    {attribute	'TcLinkTo'	:=	'.Ctrl:=TIIB[LAMP_PNL2_EP15_EP6002-0002]^COM RxPDO-Map Outputs Channel 1^Ctrl;
                                 .D[0]:=TIIB[LAMP_PNL2_EP15_EP6002-0002]^COM RxPDO-Map Outputs Channel 1^Data Out 0;
                                 .D[1]:=TIIB[LAMP_PNL2_EP15_EP6002-0002]^COM RxPDO-Map Outputs Channel 1^Data Out 1;
                                 .D[2]:=TIIB[LAMP_PNL2_EP15_EP6002-0002]^COM RxPDO-Map Outputs Channel 1^Data Out 2;
                                 .D[3]:=TIIB[LAMP_PNL2_EP15_EP6002-0002]^COM RxPDO-Map Outputs Channel 1^Data Out 3;
                                 .D[4]:=TIIB[LAMP_PNL2_EP15_EP6002-0002]^COM RxPDO-Map Outputs Channel 1^Data Out 4;
                                 .D[5]:=TIIB[LAMP_PNL2_EP15_EP6002-0002]^COM RxPDO-Map Outputs Channel 1^Data Out 5;
                                 .D[6]:=TIIB[LAMP_PNL2_EP15_EP6002-0002]^COM RxPDO-Map Outputs Channel 1^Data Out 6;
                                 .D[7]:=TIIB[LAMP_PNL2_EP15_EP6002-0002]^COM RxPDO-Map Outputs Channel 1^Data Out 7;
                                 .D[8]:=TIIB[LAMP_PNL2_EP15_EP6002-0002]^COM RxPDO-Map Outputs Channel 1^Data Out 8;
                                 .D[9]:=TIIB[LAMP_PNL2_EP15_EP6002-0002]^COM RxPDO-Map Outputs Channel 1^Data Out 9;
                                 .D[10]:=TIIB[LAMP_PNL2_EP15_EP6002-0002]^COM RxPDO-Map Outputs Channel 1^Data Out 10;
                                 .D[11]:=TIIB[LAMP_PNL2_EP15_EP6002-0002]^COM RxPDO-Map Outputs Channel 1^Data Out 11;
                                 .D[12]:=TIIB[LAMP_PNL2_EP15_EP6002-0002]^COM RxPDO-Map Outputs Channel 1^Data Out 12;
                                 .D[13]:=TIIB[LAMP_PNL2_EP15_EP6002-0002]^COM RxPDO-Map Outputs Channel 1^Data Out 13;
                                 .D[14]:=TIIB[LAMP_PNL2_EP15_EP6002-0002]^COM RxPDO-Map Outputs Channel 1^Data Out 14;
                                 .D[15]:=TIIB[LAMP_PNL2_EP15_EP6002-0002]^COM RxPDO-Map Outputs Channel 1^Data Out 15;
                                 .D[16]:=TIIB[LAMP_PNL2_EP15_EP6002-0002]^COM RxPDO-Map Outputs Channel 1^Data Out 16;
                                 .D[17]:=TIIB[LAMP_PNL2_EP15_EP6002-0002]^COM RxPDO-Map Outputs Channel 1^Data Out 17;
                                 .D[18]:=TIIB[LAMP_PNL2_EP15_EP6002-0002]^COM RxPDO-Map Outputs Channel 1^Data Out 18;
                                 .D[19]:=TIIB[LAMP_PNL2_EP15_EP6002-0002]^COM RxPDO-Map Outputs Channel 1^Data Out 19;
                                 .D[20]:=TIIB[LAMP_PNL2_EP15_EP6002-0002]^COM RxPDO-Map Outputs Channel 1^Data Out 20;
                                 .D[21]:=TIIB[LAMP_PNL2_EP15_EP6002-0002]^COM RxPDO-Map Outputs Channel 1^Data Out 21;
    '}
    stComOut_LAMP_ROUGH_PTM_01		AT %Q*	:	EL6outData22B;
(*
    {attribute	'TcLinkTo'	:=	'.Status:=TIIB[LAMP_PNL2_EP15_EP6002-0002]^COM TxPDO-Map Inputs Channel 2^Status;
                                 .D[0]:=TIIB[LAMP_PNL2_EP15_EP6002-0002]^COM TxPDO-Map Inputs Channel 2^Data In 0;
                                 .D[1]:=TIIB[LAMP_PNL2_EP15_EP6002-0002]^COM TxPDO-Map Inputs Channel 2^Data In 1;
                                 .D[2]:=TIIB[LAMP_PNL2_EP15_EP6002-0002]^COM TxPDO-Map Inputs Channel 2^Data In 2;
                                 .D[3]:=TIIB[LAMP_PNL2_EP15_EP6002-0002]^COM TxPDO-Map Inputs Channel 2^Data In 3;
                                 .D[4]:=TIIB[LAMP_PNL2_EP15_EP6002-0002]^COM TxPDO-Map Inputs Channel 2^Data In 4;
                                 .D[5]:=TIIB[LAMP_PNL2_EP15_EP6002-0002]^COM TxPDO-Map Inputs Channel 2^Data In 5;
                                 .D[6]:=TIIB[LAMP_PNL2_EP15_EP6002-0002]^COM TxPDO-Map Inputs Channel 2^Data In 6;
                                 .D[7]:=TIIB[LAMP_PNL2_EP15_EP6002-0002]^COM TxPDO-Map Inputs Channel 2^Data In 7;
                                 .D[8]:=TIIB[LAMP_PNL2_EP15_EP6002-0002]^COM TxPDO-Map Inputs Channel 2^Data In 8;
                                 .D[9]:=TIIB[LAMP_PNL2_EP15_EP6002-0002]^COM TxPDO-Map Inputs Channel 2^Data In 9;
                                 .D[10]:=TIIB[LAMP_PNL2_EP15_EP6002-0002]^COM TxPDO-Map Inputs Channel 2^Data In 10;
                                 .D[11]:=TIIB[LAMP_PNL2_EP15_EP6002-0002]^COM TxPDO-Map Inputs Channel 2^Data In 11;
                                 .D[12]:=TIIB[LAMP_PNL2_EP15_EP6002-0002]^COM TxPDO-Map Inputs Channel 2^Data In 12;
                                 .D[13]:=TIIB[LAMP_PNL2_EP15_EP6002-0002]^COM TxPDO-Map Inputs Channel 2^Data In 13;
                                 .D[14]:=TIIB[LAMP_PNL2_EP15_EP6002-0002]^COM TxPDO-Map Inputs Channel 2^Data In 14;
                                 .D[15]:=TIIB[LAMP_PNL2_EP15_EP6002-0002]^COM TxPDO-Map Inputs Channel 2^Data In 15;
                                 .D[16]:=TIIB[LAMP_PNL2_EP15_EP6002-0002]^COM TxPDO-Map Inputs Channel 2^Data In 16;
                                 .D[17]:=TIIB[LAMP_PNL2_EP15_EP6002-0002]^COM TxPDO-Map Inputs Channel 2^Data In 17;
                                 .D[18]:=TIIB[LAMP_PNL2_EP15_EP6002-0002]^COM TxPDO-Map Inputs Channel 2^Data In 18;
                                 .D[19]:=TIIB[LAMP_PNL2_EP15_EP6002-0002]^COM TxPDO-Map Inputs Channel 2^Data In 19;
                                 .D[20]:=TIIB[LAMP_PNL2_EP15_EP6002-0002]^COM TxPDO-Map Inputs Channel 2^Data In 20;
                                 .D[21]:=TIIB[LAMP_PNL2_EP15_EP6002-0002]^COM TxPDO-Map Inputs Channel 2^Data In 21;
    '}
    stComIn_LAMP_C1_PTM_01		AT %I*	:	EL6inData22B;
*)
(*
    {attribute	'TcLinkTo'	:=	'.Ctrl:=TIIB[LAMP_PNL2_EP15_EP6002-0002]^COM RxPDO-Map Outputs Channel 2^Ctrl;
                                 .D[0]:=TIIB[LAMP_PNL2_EP15_EP6002-0002]^COM RxPDO-Map Outputs Channel 2^Data Out 0;
                                 .D[1]:=TIIB[LAMP_PNL2_EP15_EP6002-0002]^COM RxPDO-Map Outputs Channel 2^Data Out 1;
                                 .D[2]:=TIIB[LAMP_PNL2_EP15_EP6002-0002]^COM RxPDO-Map Outputs Channel 2^Data Out 2;
                                 .D[3]:=TIIB[LAMP_PNL2_EP15_EP6002-0002]^COM RxPDO-Map Outputs Channel 2^Data Out 3;
                                 .D[4]:=TIIB[LAMP_PNL2_EP15_EP6002-0002]^COM RxPDO-Map Outputs Channel 2^Data Out 4;
                                 .D[5]:=TIIB[LAMP_PNL2_EP15_EP6002-0002]^COM RxPDO-Map Outputs Channel 2^Data Out 5;
                                 .D[6]:=TIIB[LAMP_PNL2_EP15_EP6002-0002]^COM RxPDO-Map Outputs Channel 2^Data Out 6;
                                 .D[7]:=TIIB[LAMP_PNL2_EP15_EP6002-0002]^COM RxPDO-Map Outputs Channel 2^Data Out 7;
                                 .D[8]:=TIIB[LAMP_PNL2_EP15_EP6002-0002]^COM RxPDO-Map Outputs Channel 2^Data Out 8;
                                 .D[9]:=TIIB[LAMP_PNL2_EP15_EP6002-0002]^COM RxPDO-Map Outputs Channel 2^Data Out 9;
                                 .D[10]:=TIIB[LAMP_PNL2_EP15_EP6002-0002]^COM RxPDO-Map Outputs Channel 2^Data Out 10;
                                 .D[11]:=TIIB[LAMP_PNL2_EP15_EP6002-0002]^COM RxPDO-Map Outputs Channel 2^Data Out 11;
                                 .D[12]:=TIIB[LAMP_PNL2_EP15_EP6002-0002]^COM RxPDO-Map Outputs Channel 2^Data Out 12;
                                 .D[13]:=TIIB[LAMP_PNL2_EP15_EP6002-0002]^COM RxPDO-Map Outputs Channel 2^Data Out 13;
                                 .D[14]:=TIIB[LAMP_PNL2_EP15_EP6002-0002]^COM RxPDO-Map Outputs Channel 2^Data Out 14;
                                 .D[15]:=TIIB[LAMP_PNL2_EP15_EP6002-0002]^COM RxPDO-Map Outputs Channel 2^Data Out 15;
                                 .D[16]:=TIIB[LAMP_PNL2_EP15_EP6002-0002]^COM RxPDO-Map Outputs Channel 2^Data Out 16;
                                 .D[17]:=TIIB[LAMP_PNL2_EP15_EP6002-0002]^COM RxPDO-Map Outputs Channel 2^Data Out 17;
                                 .D[18]:=TIIB[LAMP_PNL2_EP15_EP6002-0002]^COM RxPDO-Map Outputs Channel 2^Data Out 18;
                                 .D[19]:=TIIB[LAMP_PNL2_EP15_EP6002-0002]^COM RxPDO-Map Outputs Channel 2^Data Out 19;
                                 .D[20]:=TIIB[LAMP_PNL2_EP15_EP6002-0002]^COM RxPDO-Map Outputs Channel 2^Data Out 20;
                                 .D[21]:=TIIB[LAMP_PNL2_EP15_EP6002-0002]^COM RxPDO-Map Outputs Channel 2^Data Out 21;
    '}
    stComOut_LAMP_C1_PTM_01		AT %Q*	:	EL6outData22B;
*)
(*
    {attribute	'TcLinkTo'	:=	'.Status:=TIIB[LAMP_PNL2_EP18_EP6002-0002]^COM TxPDO-Map Inputs Channel 1^Status;
                                 .D[0]:=TIIB[LAMP_PNL2_EP18_EP6002-0002]^COM TxPDO-Map Inputs Channel 1^Data In 0;
                                 .D[1]:=TIIB[LAMP_PNL2_EP18_EP6002-0002]^COM TxPDO-Map Inputs Channel 1^Data In 1;
                                 .D[2]:=TIIB[LAMP_PNL2_EP18_EP6002-0002]^COM TxPDO-Map Inputs Channel 1^Data In 2;
                                 .D[3]:=TIIB[LAMP_PNL2_EP18_EP6002-0002]^COM TxPDO-Map Inputs Channel 1^Data In 3;
                                 .D[4]:=TIIB[LAMP_PNL2_EP18_EP6002-0002]^COM TxPDO-Map Inputs Channel 1^Data In 4;
                                 .D[5]:=TIIB[LAMP_PNL2_EP18_EP6002-0002]^COM TxPDO-Map Inputs Channel 1^Data In 5;
                                 .D[6]:=TIIB[LAMP_PNL2_EP18_EP6002-0002]^COM TxPDO-Map Inputs Channel 1^Data In 6;
                                 .D[7]:=TIIB[LAMP_PNL2_EP18_EP6002-0002]^COM TxPDO-Map Inputs Channel 1^Data In 7;
                                 .D[8]:=TIIB[LAMP_PNL2_EP18_EP6002-0002]^COM TxPDO-Map Inputs Channel 1^Data In 8;
                                 .D[9]:=TIIB[LAMP_PNL2_EP18_EP6002-0002]^COM TxPDO-Map Inputs Channel 1^Data In 9;
                                 .D[10]:=TIIB[LAMP_PNL2_EP18_EP6002-0002]^COM TxPDO-Map Inputs Channel 1^Data In 10;
                                 .D[11]:=TIIB[LAMP_PNL2_EP18_EP6002-0002]^COM TxPDO-Map Inputs Channel 1^Data In 11;
                                 .D[12]:=TIIB[LAMP_PNL2_EP18_EP6002-0002]^COM TxPDO-Map Inputs Channel 1^Data In 12;
                                 .D[13]:=TIIB[LAMP_PNL2_EP18_EP6002-0002]^COM TxPDO-Map Inputs Channel 1^Data In 13;
                                 .D[14]:=TIIB[LAMP_PNL2_EP18_EP6002-0002]^COM TxPDO-Map Inputs Channel 1^Data In 14;
                                 .D[15]:=TIIB[LAMP_PNL2_EP18_EP6002-0002]^COM TxPDO-Map Inputs Channel 1^Data In 15;
                                 .D[16]:=TIIB[LAMP_PNL2_EP18_EP6002-0002]^COM TxPDO-Map Inputs Channel 1^Data In 16;
                                 .D[17]:=TIIB[LAMP_PNL2_EP18_EP6002-0002]^COM TxPDO-Map Inputs Channel 1^Data In 17;
                                 .D[18]:=TIIB[LAMP_PNL2_EP18_EP6002-0002]^COM TxPDO-Map Inputs Channel 1^Data In 18;
                                 .D[19]:=TIIB[LAMP_PNL2_EP18_EP6002-0002]^COM TxPDO-Map Inputs Channel 1^Data In 19;
                                 .D[20]:=TIIB[LAMP_PNL2_EP18_EP6002-0002]^COM TxPDO-Map Inputs Channel 1^Data In 20;
                                 .D[21]:=TIIB[LAMP_PNL2_EP18_EP6002-0002]^COM TxPDO-Map Inputs Channel 1^Data In 21;
    '}
    stComIn_LAMP_CATCH_PTM_01		AT %I*	:	EL6inData22B;
*)
(*
    {attribute	'TcLinkTo'	:=	'.Ctrl:=TIIB[LAMP_PNL2_EP18_EP6002-0002]^COM RxPDO-Map Outputs Channel 1^Ctrl;
                                 .D[0]:=TIIB[LAMP_PNL2_EP18_EP6002-0002]^COM RxPDO-Map Outputs Channel 1^Data Out 0;
                                 .D[1]:=TIIB[LAMP_PNL2_EP18_EP6002-0002]^COM RxPDO-Map Outputs Channel 1^Data Out 1;
                                 .D[2]:=TIIB[LAMP_PNL2_EP18_EP6002-0002]^COM RxPDO-Map Outputs Channel 1^Data Out 2;
                                 .D[3]:=TIIB[LAMP_PNL2_EP18_EP6002-0002]^COM RxPDO-Map Outputs Channel 1^Data Out 3;
                                 .D[4]:=TIIB[LAMP_PNL2_EP18_EP6002-0002]^COM RxPDO-Map Outputs Channel 1^Data Out 4;
                                 .D[5]:=TIIB[LAMP_PNL2_EP18_EP6002-0002]^COM RxPDO-Map Outputs Channel 1^Data Out 5;
                                 .D[6]:=TIIB[LAMP_PNL2_EP18_EP6002-0002]^COM RxPDO-Map Outputs Channel 1^Data Out 6;
                                 .D[7]:=TIIB[LAMP_PNL2_EP18_EP6002-0002]^COM RxPDO-Map Outputs Channel 1^Data Out 7;
                                 .D[8]:=TIIB[LAMP_PNL2_EP18_EP6002-0002]^COM RxPDO-Map Outputs Channel 1^Data Out 8;
                                 .D[9]:=TIIB[LAMP_PNL2_EP18_EP6002-0002]^COM RxPDO-Map Outputs Channel 1^Data Out 9;
                                 .D[10]:=TIIB[LAMP_PNL2_EP18_EP6002-0002]^COM RxPDO-Map Outputs Channel 1^Data Out 10;
                                 .D[11]:=TIIB[LAMP_PNL2_EP18_EP6002-0002]^COM RxPDO-Map Outputs Channel 1^Data Out 11;
                                 .D[12]:=TIIB[LAMP_PNL2_EP18_EP6002-0002]^COM RxPDO-Map Outputs Channel 1^Data Out 12;
                                 .D[13]:=TIIB[LAMP_PNL2_EP18_EP6002-0002]^COM RxPDO-Map Outputs Channel 1^Data Out 13;
                                 .D[14]:=TIIB[LAMP_PNL2_EP18_EP6002-0002]^COM RxPDO-Map Outputs Channel 1^Data Out 14;
                                 .D[15]:=TIIB[LAMP_PNL2_EP18_EP6002-0002]^COM RxPDO-Map Outputs Channel 1^Data Out 15;
                                 .D[16]:=TIIB[LAMP_PNL2_EP18_EP6002-0002]^COM RxPDO-Map Outputs Channel 1^Data Out 16;
                                 .D[17]:=TIIB[LAMP_PNL2_EP18_EP6002-0002]^COM RxPDO-Map Outputs Channel 1^Data Out 17;
                                 .D[18]:=TIIB[LAMP_PNL2_EP18_EP6002-0002]^COM RxPDO-Map Outputs Channel 1^Data Out 18;
                                 .D[19]:=TIIB[LAMP_PNL2_EP18_EP6002-0002]^COM RxPDO-Map Outputs Channel 1^Data Out 19;
                                 .D[20]:=TIIB[LAMP_PNL2_EP18_EP6002-0002]^COM RxPDO-Map Outputs Channel 1^Data Out 20;
                                 .D[21]:=TIIB[LAMP_PNL2_EP18_EP6002-0002]^COM RxPDO-Map Outputs Channel 1^Data Out 21;
    '}
    stComOut_LAMP_CATCH_PTM_01		AT %Q*	:	EL6outData22B;
*)
(*
    {attribute	'TcLinkTo'	:=	'.Status:=TIIB[LAMP_PNL2_EP18_EP6002-0002]^COM TxPDO-Map Inputs Channel 2^Status;
                                 .D[0]:=TIIB[LAMP_PNL2_EP18_EP6002-0002]^COM TxPDO-Map Inputs Channel 2^Data In 0;
                                 .D[1]:=TIIB[LAMP_PNL2_EP18_EP6002-0002]^COM TxPDO-Map Inputs Channel 2^Data In 1;
                                 .D[2]:=TIIB[LAMP_PNL2_EP18_EP6002-0002]^COM TxPDO-Map Inputs Channel 2^Data In 2;
                                 .D[3]:=TIIB[LAMP_PNL2_EP18_EP6002-0002]^COM TxPDO-Map Inputs Channel 2^Data In 3;
                                 .D[4]:=TIIB[LAMP_PNL2_EP18_EP6002-0002]^COM TxPDO-Map Inputs Channel 2^Data In 4;
                                 .D[5]:=TIIB[LAMP_PNL2_EP18_EP6002-0002]^COM TxPDO-Map Inputs Channel 2^Data In 5;
                                 .D[6]:=TIIB[LAMP_PNL2_EP18_EP6002-0002]^COM TxPDO-Map Inputs Channel 2^Data In 6;
                                 .D[7]:=TIIB[LAMP_PNL2_EP18_EP6002-0002]^COM TxPDO-Map Inputs Channel 2^Data In 7;
                                 .D[8]:=TIIB[LAMP_PNL2_EP18_EP6002-0002]^COM TxPDO-Map Inputs Channel 2^Data In 8;
                                 .D[9]:=TIIB[LAMP_PNL2_EP18_EP6002-0002]^COM TxPDO-Map Inputs Channel 2^Data In 9;
                                 .D[10]:=TIIB[LAMP_PNL2_EP18_EP6002-0002]^COM TxPDO-Map Inputs Channel 2^Data In 10;
                                 .D[11]:=TIIB[LAMP_PNL2_EP18_EP6002-0002]^COM TxPDO-Map Inputs Channel 2^Data In 11;
                                 .D[12]:=TIIB[LAMP_PNL2_EP18_EP6002-0002]^COM TxPDO-Map Inputs Channel 2^Data In 12;
                                 .D[13]:=TIIB[LAMP_PNL2_EP18_EP6002-0002]^COM TxPDO-Map Inputs Channel 2^Data In 13;
                                 .D[14]:=TIIB[LAMP_PNL2_EP18_EP6002-0002]^COM TxPDO-Map Inputs Channel 2^Data In 14;
                                 .D[15]:=TIIB[LAMP_PNL2_EP18_EP6002-0002]^COM TxPDO-Map Inputs Channel 2^Data In 15;
                                 .D[16]:=TIIB[LAMP_PNL2_EP18_EP6002-0002]^COM TxPDO-Map Inputs Channel 2^Data In 16;
                                 .D[17]:=TIIB[LAMP_PNL2_EP18_EP6002-0002]^COM TxPDO-Map Inputs Channel 2^Data In 17;
                                 .D[18]:=TIIB[LAMP_PNL2_EP18_EP6002-0002]^COM TxPDO-Map Inputs Channel 2^Data In 18;
                                 .D[19]:=TIIB[LAMP_PNL2_EP18_EP6002-0002]^COM TxPDO-Map Inputs Channel 2^Data In 19;
                                 .D[20]:=TIIB[LAMP_PNL2_EP18_EP6002-0002]^COM TxPDO-Map Inputs Channel 2^Data In 20;
                                 .D[21]:=TIIB[LAMP_PNL2_EP18_EP6002-0002]^COM TxPDO-Map Inputs Channel 2^Data In 21;
    '}
    stComIn_LAMP_CATCH_PTM_02		AT %I*	:	EL6inData22B;
*)
(*
    {attribute	'TcLinkTo'	:=	'.Ctrl:=TIIB[LAMP_PNL2_EP18_EP6002-0002]^COM RxPDO-Map Outputs Channel 2^Ctrl;
                                 .D[0]:=TIIB[LAMP_PNL2_EP18_EP6002-0002]^COM RxPDO-Map Outputs Channel 2^Data Out 0;
                                 .D[1]:=TIIB[LAMP_PNL2_EP18_EP6002-0002]^COM RxPDO-Map Outputs Channel 2^Data Out 1;
                                 .D[2]:=TIIB[LAMP_PNL2_EP18_EP6002-0002]^COM RxPDO-Map Outputs Channel 2^Data Out 2;
                                 .D[3]:=TIIB[LAMP_PNL2_EP18_EP6002-0002]^COM RxPDO-Map Outputs Channel 2^Data Out 3;
                                 .D[4]:=TIIB[LAMP_PNL2_EP18_EP6002-0002]^COM RxPDO-Map Outputs Channel 2^Data Out 4;
                                 .D[5]:=TIIB[LAMP_PNL2_EP18_EP6002-0002]^COM RxPDO-Map Outputs Channel 2^Data Out 5;
                                 .D[6]:=TIIB[LAMP_PNL2_EP18_EP6002-0002]^COM RxPDO-Map Outputs Channel 2^Data Out 6;
                                 .D[7]:=TIIB[LAMP_PNL2_EP18_EP6002-0002]^COM RxPDO-Map Outputs Channel 2^Data Out 7;
                                 .D[8]:=TIIB[LAMP_PNL2_EP18_EP6002-0002]^COM RxPDO-Map Outputs Channel 2^Data Out 8;
                                 .D[9]:=TIIB[LAMP_PNL2_EP18_EP6002-0002]^COM RxPDO-Map Outputs Channel 2^Data Out 9;
                                 .D[10]:=TIIB[LAMP_PNL2_EP18_EP6002-0002]^COM RxPDO-Map Outputs Channel 2^Data Out 10;
                                 .D[11]:=TIIB[LAMP_PNL2_EP18_EP6002-0002]^COM RxPDO-Map Outputs Channel 2^Data Out 11;
                                 .D[12]:=TIIB[LAMP_PNL2_EP18_EP6002-0002]^COM RxPDO-Map Outputs Channel 2^Data Out 12;
                                 .D[13]:=TIIB[LAMP_PNL2_EP18_EP6002-0002]^COM RxPDO-Map Outputs Channel 2^Data Out 13;
                                 .D[14]:=TIIB[LAMP_PNL2_EP18_EP6002-0002]^COM RxPDO-Map Outputs Channel 2^Data Out 14;
                                 .D[15]:=TIIB[LAMP_PNL2_EP18_EP6002-0002]^COM RxPDO-Map Outputs Channel 2^Data Out 15;
                                 .D[16]:=TIIB[LAMP_PNL2_EP18_EP6002-0002]^COM RxPDO-Map Outputs Channel 2^Data Out 16;
                                 .D[17]:=TIIB[LAMP_PNL2_EP18_EP6002-0002]^COM RxPDO-Map Outputs Channel 2^Data Out 17;
                                 .D[18]:=TIIB[LAMP_PNL2_EP18_EP6002-0002]^COM RxPDO-Map Outputs Channel 2^Data Out 18;
                                 .D[19]:=TIIB[LAMP_PNL2_EP18_EP6002-0002]^COM RxPDO-Map Outputs Channel 2^Data Out 19;
                                 .D[20]:=TIIB[LAMP_PNL2_EP18_EP6002-0002]^COM RxPDO-Map Outputs Channel 2^Data Out 20;
                                 .D[21]:=TIIB[LAMP_PNL2_EP18_EP6002-0002]^COM RxPDO-Map Outputs Channel 2^Data Out 21;
    '}
    stComOut_LAMP_CATCH_PTM_02		AT %Q*	:	EL6outData22B;
*)
(*
    {attribute	'TcLinkTo'	:=	'.Status:=TIIB[KTOF_PNL1_EP03_EP6002-0002]^COM TxPDO-Map Inputs Channel 1^Status;
                                 .D[0]:=TIIB[KTOF_PNL1_EP03_EP6002-0002]^COM TxPDO-Map Inputs Channel 1^Data In 0;
                                 .D[1]:=TIIB[KTOF_PNL1_EP03_EP6002-0002]^COM TxPDO-Map Inputs Channel 1^Data In 1;
                                 .D[2]:=TIIB[KTOF_PNL1_EP03_EP6002-0002]^COM TxPDO-Map Inputs Channel 1^Data In 2;
                                 .D[3]:=TIIB[KTOF_PNL1_EP03_EP6002-0002]^COM TxPDO-Map Inputs Channel 1^Data In 3;
                                 .D[4]:=TIIB[KTOF_PNL1_EP03_EP6002-0002]^COM TxPDO-Map Inputs Channel 1^Data In 4;
                                 .D[5]:=TIIB[KTOF_PNL1_EP03_EP6002-0002]^COM TxPDO-Map Inputs Channel 1^Data In 5;
                                 .D[6]:=TIIB[KTOF_PNL1_EP03_EP6002-0002]^COM TxPDO-Map Inputs Channel 1^Data In 6;
                                 .D[7]:=TIIB[KTOF_PNL1_EP03_EP6002-0002]^COM TxPDO-Map Inputs Channel 1^Data In 7;
                                 .D[8]:=TIIB[KTOF_PNL1_EP03_EP6002-0002]^COM TxPDO-Map Inputs Channel 1^Data In 8;
                                 .D[9]:=TIIB[KTOF_PNL1_EP03_EP6002-0002]^COM TxPDO-Map Inputs Channel 1^Data In 9;
                                 .D[10]:=TIIB[KTOF_PNL1_EP03_EP6002-0002]^COM TxPDO-Map Inputs Channel 1^Data In 10;
                                 .D[11]:=TIIB[KTOF_PNL1_EP03_EP6002-0002]^COM TxPDO-Map Inputs Channel 1^Data In 11;
                                 .D[12]:=TIIB[KTOF_PNL1_EP03_EP6002-0002]^COM TxPDO-Map Inputs Channel 1^Data In 12;
                                 .D[13]:=TIIB[KTOF_PNL1_EP03_EP6002-0002]^COM TxPDO-Map Inputs Channel 1^Data In 13;
                                 .D[14]:=TIIB[KTOF_PNL1_EP03_EP6002-0002]^COM TxPDO-Map Inputs Channel 1^Data In 14;
                                 .D[15]:=TIIB[KTOF_PNL1_EP03_EP6002-0002]^COM TxPDO-Map Inputs Channel 1^Data In 15;
                                 .D[16]:=TIIB[KTOF_PNL1_EP03_EP6002-0002]^COM TxPDO-Map Inputs Channel 1^Data In 16;
                                 .D[17]:=TIIB[KTOF_PNL1_EP03_EP6002-0002]^COM TxPDO-Map Inputs Channel 1^Data In 17;
                                 .D[18]:=TIIB[KTOF_PNL1_EP03_EP6002-0002]^COM TxPDO-Map Inputs Channel 1^Data In 18;
                                 .D[19]:=TIIB[KTOF_PNL1_EP03_EP6002-0002]^COM TxPDO-Map Inputs Channel 1^Data In 19;
                                 .D[20]:=TIIB[KTOF_PNL1_EP03_EP6002-0002]^COM TxPDO-Map Inputs Channel 1^Data In 20;
                                 .D[21]:=TIIB[KTOF_PNL1_EP03_EP6002-0002]^COM TxPDO-Map Inputs Channel 1^Data In 21;
    '}
    stComIn_KTOF_PTM_01		AT %I*	:	EL6inData22B;
*)
(*
    {attribute	'TcLinkTo'	:=	'.Ctrl:=TIIB[KTOF_PNL1_EP03_EP6002-0002]^COM RxPDO-Map Outputs Channel 1^Ctrl;
                                 .D[0]:=TIIB[KTOF_PNL1_EP03_EP6002-0002]^COM RxPDO-Map Outputs Channel 1^Data Out 0;
                                 .D[1]:=TIIB[KTOF_PNL1_EP03_EP6002-0002]^COM RxPDO-Map Outputs Channel 1^Data Out 1;
                                 .D[2]:=TIIB[KTOF_PNL1_EP03_EP6002-0002]^COM RxPDO-Map Outputs Channel 1^Data Out 2;
                                 .D[3]:=TIIB[KTOF_PNL1_EP03_EP6002-0002]^COM RxPDO-Map Outputs Channel 1^Data Out 3;
                                 .D[4]:=TIIB[KTOF_PNL1_EP03_EP6002-0002]^COM RxPDO-Map Outputs Channel 1^Data Out 4;
                                 .D[5]:=TIIB[KTOF_PNL1_EP03_EP6002-0002]^COM RxPDO-Map Outputs Channel 1^Data Out 5;
                                 .D[6]:=TIIB[KTOF_PNL1_EP03_EP6002-0002]^COM RxPDO-Map Outputs Channel 1^Data Out 6;
                                 .D[7]:=TIIB[KTOF_PNL1_EP03_EP6002-0002]^COM RxPDO-Map Outputs Channel 1^Data Out 7;
                                 .D[8]:=TIIB[KTOF_PNL1_EP03_EP6002-0002]^COM RxPDO-Map Outputs Channel 1^Data Out 8;
                                 .D[9]:=TIIB[KTOF_PNL1_EP03_EP6002-0002]^COM RxPDO-Map Outputs Channel 1^Data Out 9;
                                 .D[10]:=TIIB[KTOF_PNL1_EP03_EP6002-0002]^COM RxPDO-Map Outputs Channel 1^Data Out 10;
                                 .D[11]:=TIIB[KTOF_PNL1_EP03_EP6002-0002]^COM RxPDO-Map Outputs Channel 1^Data Out 11;
                                 .D[12]:=TIIB[KTOF_PNL1_EP03_EP6002-0002]^COM RxPDO-Map Outputs Channel 1^Data Out 12;
                                 .D[13]:=TIIB[KTOF_PNL1_EP03_EP6002-0002]^COM RxPDO-Map Outputs Channel 1^Data Out 13;
                                 .D[14]:=TIIB[KTOF_PNL1_EP03_EP6002-0002]^COM RxPDO-Map Outputs Channel 1^Data Out 14;
                                 .D[15]:=TIIB[KTOF_PNL1_EP03_EP6002-0002]^COM RxPDO-Map Outputs Channel 1^Data Out 15;
                                 .D[16]:=TIIB[KTOF_PNL1_EP03_EP6002-0002]^COM RxPDO-Map Outputs Channel 1^Data Out 16;
                                 .D[17]:=TIIB[KTOF_PNL1_EP03_EP6002-0002]^COM RxPDO-Map Outputs Channel 1^Data Out 17;
                                 .D[18]:=TIIB[KTOF_PNL1_EP03_EP6002-0002]^COM RxPDO-Map Outputs Channel 1^Data Out 18;
                                 .D[19]:=TIIB[KTOF_PNL1_EP03_EP6002-0002]^COM RxPDO-Map Outputs Channel 1^Data Out 19;
                                 .D[20]:=TIIB[KTOF_PNL1_EP03_EP6002-0002]^COM RxPDO-Map Outputs Channel 1^Data Out 20;
                                 .D[21]:=TIIB[KTOF_PNL1_EP03_EP6002-0002]^COM RxPDO-Map Outputs Channel 1^Data Out 21;
    '}
    stComOut_KTOF_PTM_01		AT %Q*	:	EL6outData22B;
*)
    //Leybolds
    {attribute	'TcLinkTo'	:=	'.Status:=TIIB[LAMP_PLC_E11_EL6002]^COM TxPDO-Map Inputs Channel 1^Status;
                                 .D[0]:=TIIB[LAMP_PLC_E11_EL6002]^COM TxPDO-Map Inputs Channel 1^Data In 0;
                                 .D[1]:=TIIB[LAMP_PLC_E11_EL6002]^COM TxPDO-Map Inputs Channel 1^Data In 1;
                                 .D[2]:=TIIB[LAMP_PLC_E11_EL6002]^COM TxPDO-Map Inputs Channel 1^Data In 2;
                                 .D[3]:=TIIB[LAMP_PLC_E11_EL6002]^COM TxPDO-Map Inputs Channel 1^Data In 3;
                                 .D[4]:=TIIB[LAMP_PLC_E11_EL6002]^COM TxPDO-Map Inputs Channel 1^Data In 4;
                                 .D[5]:=TIIB[LAMP_PLC_E11_EL6002]^COM TxPDO-Map Inputs Channel 1^Data In 5;
                                 .D[6]:=TIIB[LAMP_PLC_E11_EL6002]^COM TxPDO-Map Inputs Channel 1^Data In 6;
                                 .D[7]:=TIIB[LAMP_PLC_E11_EL6002]^COM TxPDO-Map Inputs Channel 1^Data In 7;
                                 .D[8]:=TIIB[LAMP_PLC_E11_EL6002]^COM TxPDO-Map Inputs Channel 1^Data In 8;
                                 .D[9]:=TIIB[LAMP_PLC_E11_EL6002]^COM TxPDO-Map Inputs Channel 1^Data In 9;
                                 .D[10]:=TIIB[LAMP_PLC_E11_EL6002]^COM TxPDO-Map Inputs Channel 1^Data In 10;
                                 .D[11]:=TIIB[LAMP_PLC_E11_EL6002]^COM TxPDO-Map Inputs Channel 1^Data In 11;
                                 .D[12]:=TIIB[LAMP_PLC_E11_EL6002]^COM TxPDO-Map Inputs Channel 1^Data In 12;
                                 .D[13]:=TIIB[LAMP_PLC_E11_EL6002]^COM TxPDO-Map Inputs Channel 1^Data In 13;
                                 .D[14]:=TIIB[LAMP_PLC_E11_EL6002]^COM TxPDO-Map Inputs Channel 1^Data In 14;
                                 .D[15]:=TIIB[LAMP_PLC_E11_EL6002]^COM TxPDO-Map Inputs Channel 1^Data In 15;
                                 .D[16]:=TIIB[LAMP_PLC_E11_EL6002]^COM TxPDO-Map Inputs Channel 1^Data In 16;
                                 .D[17]:=TIIB[LAMP_PLC_E11_EL6002]^COM TxPDO-Map Inputs Channel 1^Data In 17;
                                 .D[18]:=TIIB[LAMP_PLC_E11_EL6002]^COM TxPDO-Map Inputs Channel 1^Data In 18;
                                 .D[19]:=TIIB[LAMP_PLC_E11_EL6002]^COM TxPDO-Map Inputs Channel 1^Data In 19;
                                 .D[20]:=TIIB[LAMP_PLC_E11_EL6002]^COM TxPDO-Map Inputs Channel 1^Data In 20;
                                 .D[21]:=TIIB[LAMP_PLC_E11_EL6002]^COM TxPDO-Map Inputs Channel 1^Data In 21;
    '}
    stComIn_LAMP_GJ2_PTM_01		AT %I*	:	EL6inData22B;

    {attribute	'TcLinkTo'	:=	'.Ctrl:=TIIB[LAMP_PLC_E11_EL6002]^COM RxPDO-Map Outputs Channel 1^Ctrl;
                                 .D[0]:=TIIB[LAMP_PLC_E11_EL6002]^COM RxPDO-Map Outputs Channel 1^Data Out 0;
                                 .D[1]:=TIIB[LAMP_PLC_E11_EL6002]^COM RxPDO-Map Outputs Channel 1^Data Out 1;
                                 .D[2]:=TIIB[LAMP_PLC_E11_EL6002]^COM RxPDO-Map Outputs Channel 1^Data Out 2;
                                 .D[3]:=TIIB[LAMP_PLC_E11_EL6002]^COM RxPDO-Map Outputs Channel 1^Data Out 3;
                                 .D[4]:=TIIB[LAMP_PLC_E11_EL6002]^COM RxPDO-Map Outputs Channel 1^Data Out 4;
                                 .D[5]:=TIIB[LAMP_PLC_E11_EL6002]^COM RxPDO-Map Outputs Channel 1^Data Out 5;
                                 .D[6]:=TIIB[LAMP_PLC_E11_EL6002]^COM RxPDO-Map Outputs Channel 1^Data Out 6;
                                 .D[7]:=TIIB[LAMP_PLC_E11_EL6002]^COM RxPDO-Map Outputs Channel 1^Data Out 7;
                                 .D[8]:=TIIB[LAMP_PLC_E11_EL6002]^COM RxPDO-Map Outputs Channel 1^Data Out 8;
                                 .D[9]:=TIIB[LAMP_PLC_E11_EL6002]^COM RxPDO-Map Outputs Channel 1^Data Out 9;
                                 .D[10]:=TIIB[LAMP_PLC_E11_EL6002]^COM RxPDO-Map Outputs Channel 1^Data Out 10;
                                 .D[11]:=TIIB[LAMP_PLC_E11_EL6002]^COM RxPDO-Map Outputs Channel 1^Data Out 11;
                                 .D[12]:=TIIB[LAMP_PLC_E11_EL6002]^COM RxPDO-Map Outputs Channel 1^Data Out 12;
                                 .D[13]:=TIIB[LAMP_PLC_E11_EL6002]^COM RxPDO-Map Outputs Channel 1^Data Out 13;
                                 .D[14]:=TIIB[LAMP_PLC_E11_EL6002]^COM RxPDO-Map Outputs Channel 1^Data Out 14;
                                 .D[15]:=TIIB[LAMP_PLC_E11_EL6002]^COM RxPDO-Map Outputs Channel 1^Data Out 15;
                                 .D[16]:=TIIB[LAMP_PLC_E11_EL6002]^COM RxPDO-Map Outputs Channel 1^Data Out 16;
                                 .D[17]:=TIIB[LAMP_PLC_E11_EL6002]^COM RxPDO-Map Outputs Channel 1^Data Out 17;
                                 .D[18]:=TIIB[LAMP_PLC_E11_EL6002]^COM RxPDO-Map Outputs Channel 1^Data Out 18;
                                 .D[19]:=TIIB[LAMP_PLC_E11_EL6002]^COM RxPDO-Map Outputs Channel 1^Data Out 19;
                                 .D[20]:=TIIB[LAMP_PLC_E11_EL6002]^COM RxPDO-Map Outputs Channel 1^Data Out 20;
                                 .D[21]:=TIIB[LAMP_PLC_E11_EL6002]^COM RxPDO-Map Outputs Channel 1^Data Out 21;
    '}
    stComOut_LAMP_GJ2_PTM_01		AT %Q*	:	EL6outData22B;
(*
    {attribute	'TcLinkTo'	:=	'.Status:=TIIB[LAMP_PLC_E11_EL6002]^COM TxPDO-Map Inputs Channel 2^Status;
                                 .D[0]:=TIIB[LAMP_PLC_E11_EL6002]^COM TxPDO-Map Inputs Channel 2^Data In 0;
                                 .D[1]:=TIIB[LAMP_PLC_E11_EL6002]^COM TxPDO-Map Inputs Channel 2^Data In 1;
                                 .D[2]:=TIIB[LAMP_PLC_E11_EL6002]^COM TxPDO-Map Inputs Channel 2^Data In 2;
                                 .D[3]:=TIIB[LAMP_PLC_E11_EL6002]^COM TxPDO-Map Inputs Channel 2^Data In 3;
                                 .D[4]:=TIIB[LAMP_PLC_E11_EL6002]^COM TxPDO-Map Inputs Channel 2^Data In 4;
                                 .D[5]:=TIIB[LAMP_PLC_E11_EL6002]^COM TxPDO-Map Inputs Channel 2^Data In 5;
                                 .D[6]:=TIIB[LAMP_PLC_E11_EL6002]^COM TxPDO-Map Inputs Channel 2^Data In 6;
                                 .D[7]:=TIIB[LAMP_PLC_E11_EL6002]^COM TxPDO-Map Inputs Channel 2^Data In 7;
                                 .D[8]:=TIIB[LAMP_PLC_E11_EL6002]^COM TxPDO-Map Inputs Channel 2^Data In 8;
                                 .D[9]:=TIIB[LAMP_PLC_E11_EL6002]^COM TxPDO-Map Inputs Channel 2^Data In 9;
                                 .D[10]:=TIIB[LAMP_PLC_E11_EL6002]^COM TxPDO-Map Inputs Channel 2^Data In 10;
                                 .D[11]:=TIIB[LAMP_PLC_E11_EL6002]^COM TxPDO-Map Inputs Channel 2^Data In 11;
                                 .D[12]:=TIIB[LAMP_PLC_E11_EL6002]^COM TxPDO-Map Inputs Channel 2^Data In 12;
                                 .D[13]:=TIIB[LAMP_PLC_E11_EL6002]^COM TxPDO-Map Inputs Channel 2^Data In 13;
                                 .D[14]:=TIIB[LAMP_PLC_E11_EL6002]^COM TxPDO-Map Inputs Channel 2^Data In 14;
                                 .D[15]:=TIIB[LAMP_PLC_E11_EL6002]^COM TxPDO-Map Inputs Channel 2^Data In 15;
                                 .D[16]:=TIIB[LAMP_PLC_E11_EL6002]^COM TxPDO-Map Inputs Channel 2^Data In 16;
                                 .D[17]:=TIIB[LAMP_PLC_E11_EL6002]^COM TxPDO-Map Inputs Channel 2^Data In 17;
                                 .D[18]:=TIIB[LAMP_PLC_E11_EL6002]^COM TxPDO-Map Inputs Channel 2^Data In 18;
                                 .D[19]:=TIIB[LAMP_PLC_E11_EL6002]^COM TxPDO-Map Inputs Channel 2^Data In 19;
                                 .D[20]:=TIIB[LAMP_PLC_E11_EL6002]^COM TxPDO-Map Inputs Channel 2^Data In 20;
                                 .D[21]:=TIIB[LAMP_PLC_E11_EL6002]^COM TxPDO-Map Inputs Channel 2^Data In 21;
    '}
    stComIn_LAMP_GJ2_PTM_02		AT %I*	:	EL6inData22B;
*)
(*
    {attribute	'TcLinkTo'	:=	'.Ctrl:=TIIB[LAMP_PLC_E11_EL6002]^COM RxPDO-Map Outputs Channel 2^Ctrl;
                                 .D[0]:=TIIB[LAMP_PLC_E11_EL6002]^COM RxPDO-Map Outputs Channel 2^Data Out 0;
                                 .D[1]:=TIIB[LAMP_PLC_E11_EL6002]^COM RxPDO-Map Outputs Channel 2^Data Out 1;
                                 .D[2]:=TIIB[LAMP_PLC_E11_EL6002]^COM RxPDO-Map Outputs Channel 2^Data Out 2;
                                 .D[3]:=TIIB[LAMP_PLC_E11_EL6002]^COM RxPDO-Map Outputs Channel 2^Data Out 3;
                                 .D[4]:=TIIB[LAMP_PLC_E11_EL6002]^COM RxPDO-Map Outputs Channel 2^Data Out 4;
                                 .D[5]:=TIIB[LAMP_PLC_E11_EL6002]^COM RxPDO-Map Outputs Channel 2^Data Out 5;
                                 .D[6]:=TIIB[LAMP_PLC_E11_EL6002]^COM RxPDO-Map Outputs Channel 2^Data Out 6;
                                 .D[7]:=TIIB[LAMP_PLC_E11_EL6002]^COM RxPDO-Map Outputs Channel 2^Data Out 7;
                                 .D[8]:=TIIB[LAMP_PLC_E11_EL6002]^COM RxPDO-Map Outputs Channel 2^Data Out 8;
                                 .D[9]:=TIIB[LAMP_PLC_E11_EL6002]^COM RxPDO-Map Outputs Channel 2^Data Out 9;
                                 .D[10]:=TIIB[LAMP_PLC_E11_EL6002]^COM RxPDO-Map Outputs Channel 2^Data Out 10;
                                 .D[11]:=TIIB[LAMP_PLC_E11_EL6002]^COM RxPDO-Map Outputs Channel 2^Data Out 11;
                                 .D[12]:=TIIB[LAMP_PLC_E11_EL6002]^COM RxPDO-Map Outputs Channel 2^Data Out 12;
                                 .D[13]:=TIIB[LAMP_PLC_E11_EL6002]^COM RxPDO-Map Outputs Channel 2^Data Out 13;
                                 .D[14]:=TIIB[LAMP_PLC_E11_EL6002]^COM RxPDO-Map Outputs Channel 2^Data Out 14;
                                 .D[15]:=TIIB[LAMP_PLC_E11_EL6002]^COM RxPDO-Map Outputs Channel 2^Data Out 15;
                                 .D[16]:=TIIB[LAMP_PLC_E11_EL6002]^COM RxPDO-Map Outputs Channel 2^Data Out 16;
                                 .D[17]:=TIIB[LAMP_PLC_E11_EL6002]^COM RxPDO-Map Outputs Channel 2^Data Out 17;
                                 .D[18]:=TIIB[LAMP_PLC_E11_EL6002]^COM RxPDO-Map Outputs Channel 2^Data Out 18;
                                 .D[19]:=TIIB[LAMP_PLC_E11_EL6002]^COM RxPDO-Map Outputs Channel 2^Data Out 19;
                                 .D[20]:=TIIB[LAMP_PLC_E11_EL6002]^COM RxPDO-Map Outputs Channel 2^Data Out 20;
                                 .D[21]:=TIIB[LAMP_PLC_E11_EL6002]^COM RxPDO-Map Outputs Channel 2^Data Out 21;
    '}
    stComOut_LAMP_GJ2_PTM_02		AT %Q*	:	EL6outData22B;
*)
(*
    {attribute	'TcLinkTo'	:=	'.Status:=TIIB[LAMP_PLC_E12_EL6002]^COM TxPDO-Map Inputs Channel 1^Status;
                                 .D[0]:=TIIB[LAMP_PLC_E12_EL6002]^COM TxPDO-Map Inputs Channel 1^Data In 0;
                                 .D[1]:=TIIB[LAMP_PLC_E12_EL6002]^COM TxPDO-Map Inputs Channel 1^Data In 1;
                                 .D[2]:=TIIB[LAMP_PLC_E12_EL6002]^COM TxPDO-Map Inputs Channel 1^Data In 2;
                                 .D[3]:=TIIB[LAMP_PLC_E12_EL6002]^COM TxPDO-Map Inputs Channel 1^Data In 3;
                                 .D[4]:=TIIB[LAMP_PLC_E12_EL6002]^COM TxPDO-Map Inputs Channel 1^Data In 4;
                                 .D[5]:=TIIB[LAMP_PLC_E12_EL6002]^COM TxPDO-Map Inputs Channel 1^Data In 5;
                                 .D[6]:=TIIB[LAMP_PLC_E12_EL6002]^COM TxPDO-Map Inputs Channel 1^Data In 6;
                                 .D[7]:=TIIB[LAMP_PLC_E12_EL6002]^COM TxPDO-Map Inputs Channel 1^Data In 7;
                                 .D[8]:=TIIB[LAMP_PLC_E12_EL6002]^COM TxPDO-Map Inputs Channel 1^Data In 8;
                                 .D[9]:=TIIB[LAMP_PLC_E12_EL6002]^COM TxPDO-Map Inputs Channel 1^Data In 9;
                                 .D[10]:=TIIB[LAMP_PLC_E12_EL6002]^COM TxPDO-Map Inputs Channel 1^Data In 10;
                                 .D[11]:=TIIB[LAMP_PLC_E12_EL6002]^COM TxPDO-Map Inputs Channel 1^Data In 11;
                                 .D[12]:=TIIB[LAMP_PLC_E12_EL6002]^COM TxPDO-Map Inputs Channel 1^Data In 12;
                                 .D[13]:=TIIB[LAMP_PLC_E12_EL6002]^COM TxPDO-Map Inputs Channel 1^Data In 13;
                                 .D[14]:=TIIB[LAMP_PLC_E12_EL6002]^COM TxPDO-Map Inputs Channel 1^Data In 14;
                                 .D[15]:=TIIB[LAMP_PLC_E12_EL6002]^COM TxPDO-Map Inputs Channel 1^Data In 15;
                                 .D[16]:=TIIB[LAMP_PLC_E12_EL6002]^COM TxPDO-Map Inputs Channel 1^Data In 16;
                                 .D[17]:=TIIB[LAMP_PLC_E12_EL6002]^COM TxPDO-Map Inputs Channel 1^Data In 17;
                                 .D[18]:=TIIB[LAMP_PLC_E12_EL6002]^COM TxPDO-Map Inputs Channel 1^Data In 18;
                                 .D[19]:=TIIB[LAMP_PLC_E12_EL6002]^COM TxPDO-Map Inputs Channel 1^Data In 19;
                                 .D[20]:=TIIB[LAMP_PLC_E12_EL6002]^COM TxPDO-Map Inputs Channel 1^Data In 20;
                                 .D[21]:=TIIB[LAMP_PLC_E12_EL6002]^COM TxPDO-Map Inputs Channel 1^Data In 21;
    '}
    stComIn_LAMP_GJ2_PTM_03		AT %I*	:	EL6inData22B;
*)
(*
    {attribute	'TcLinkTo'	:=	'.Ctrl:=TIIB[LAMP_PLC_E12_EL6002]^COM RxPDO-Map Outputs Channel 1^Ctrl;
                                 .D[0]:=TIIB[LAMP_PLC_E12_EL6002]^COM RxPDO-Map Outputs Channel 1^Data Out 0;
                                 .D[1]:=TIIB[LAMP_PLC_E12_EL6002]^COM RxPDO-Map Outputs Channel 1^Data Out 1;
                                 .D[2]:=TIIB[LAMP_PLC_E12_EL6002]^COM RxPDO-Map Outputs Channel 1^Data Out 2;
                                 .D[3]:=TIIB[LAMP_PLC_E12_EL6002]^COM RxPDO-Map Outputs Channel 1^Data Out 3;
                                 .D[4]:=TIIB[LAMP_PLC_E12_EL6002]^COM RxPDO-Map Outputs Channel 1^Data Out 4;
                                 .D[5]:=TIIB[LAMP_PLC_E12_EL6002]^COM RxPDO-Map Outputs Channel 1^Data Out 5;
                                 .D[6]:=TIIB[LAMP_PLC_E12_EL6002]^COM RxPDO-Map Outputs Channel 1^Data Out 6;
                                 .D[7]:=TIIB[LAMP_PLC_E12_EL6002]^COM RxPDO-Map Outputs Channel 1^Data Out 7;
                                 .D[8]:=TIIB[LAMP_PLC_E12_EL6002]^COM RxPDO-Map Outputs Channel 1^Data Out 8;
                                 .D[9]:=TIIB[LAMP_PLC_E12_EL6002]^COM RxPDO-Map Outputs Channel 1^Data Out 9;
                                 .D[10]:=TIIB[LAMP_PLC_E12_EL6002]^COM RxPDO-Map Outputs Channel 1^Data Out 10;
                                 .D[11]:=TIIB[LAMP_PLC_E12_EL6002]^COM RxPDO-Map Outputs Channel 1^Data Out 11;
                                 .D[12]:=TIIB[LAMP_PLC_E12_EL6002]^COM RxPDO-Map Outputs Channel 1^Data Out 12;
                                 .D[13]:=TIIB[LAMP_PLC_E12_EL6002]^COM RxPDO-Map Outputs Channel 1^Data Out 13;
                                 .D[14]:=TIIB[LAMP_PLC_E12_EL6002]^COM RxPDO-Map Outputs Channel 1^Data Out 14;
                                 .D[15]:=TIIB[LAMP_PLC_E12_EL6002]^COM RxPDO-Map Outputs Channel 1^Data Out 15;
                                 .D[16]:=TIIB[LAMP_PLC_E12_EL6002]^COM RxPDO-Map Outputs Channel 1^Data Out 16;
                                 .D[17]:=TIIB[LAMP_PLC_E12_EL6002]^COM RxPDO-Map Outputs Channel 1^Data Out 17;
                                 .D[18]:=TIIB[LAMP_PLC_E12_EL6002]^COM RxPDO-Map Outputs Channel 1^Data Out 18;
                                 .D[19]:=TIIB[LAMP_PLC_E12_EL6002]^COM RxPDO-Map Outputs Channel 1^Data Out 19;
                                 .D[20]:=TIIB[LAMP_PLC_E12_EL6002]^COM RxPDO-Map Outputs Channel 1^Data Out 20;
                                 .D[21]:=TIIB[LAMP_PLC_E12_EL6002]^COM RxPDO-Map Outputs Channel 1^Data Out 21;
    '}
    stComOut_LAMP_GJ2_PTM_03		AT %Q*	:	EL6outData22B;
*)
(*
    {attribute	'TcLinkTo'	:=	'.Status:=TIIB[LAMP_PLC_E12_EL6002]^COM TxPDO-Map Inputs Channel 2^Status;
                                 .D[0]:=TIIB[LAMP_PLC_E12_EL6002]^COM TxPDO-Map Inputs Channel 2^Data In 0;
                                 .D[1]:=TIIB[LAMP_PLC_E12_EL6002]^COM TxPDO-Map Inputs Channel 2^Data In 1;
                                 .D[2]:=TIIB[LAMP_PLC_E12_EL6002]^COM TxPDO-Map Inputs Channel 2^Data In 2;
                                 .D[3]:=TIIB[LAMP_PLC_E12_EL6002]^COM TxPDO-Map Inputs Channel 2^Data In 3;
                                 .D[4]:=TIIB[LAMP_PLC_E12_EL6002]^COM TxPDO-Map Inputs Channel 2^Data In 4;
                                 .D[5]:=TIIB[LAMP_PLC_E12_EL6002]^COM TxPDO-Map Inputs Channel 2^Data In 5;
                                 .D[6]:=TIIB[LAMP_PLC_E12_EL6002]^COM TxPDO-Map Inputs Channel 2^Data In 6;
                                 .D[7]:=TIIB[LAMP_PLC_E12_EL6002]^COM TxPDO-Map Inputs Channel 2^Data In 7;
                                 .D[8]:=TIIB[LAMP_PLC_E12_EL6002]^COM TxPDO-Map Inputs Channel 2^Data In 8;
                                 .D[9]:=TIIB[LAMP_PLC_E12_EL6002]^COM TxPDO-Map Inputs Channel 2^Data In 9;
                                 .D[10]:=TIIB[LAMP_PLC_E12_EL6002]^COM TxPDO-Map Inputs Channel 2^Data In 10;
                                 .D[11]:=TIIB[LAMP_PLC_E12_EL6002]^COM TxPDO-Map Inputs Channel 2^Data In 11;
                                 .D[12]:=TIIB[LAMP_PLC_E12_EL6002]^COM TxPDO-Map Inputs Channel 2^Data In 12;
                                 .D[13]:=TIIB[LAMP_PLC_E12_EL6002]^COM TxPDO-Map Inputs Channel 2^Data In 13;
                                 .D[14]:=TIIB[LAMP_PLC_E12_EL6002]^COM TxPDO-Map Inputs Channel 2^Data In 14;
                                 .D[15]:=TIIB[LAMP_PLC_E12_EL6002]^COM TxPDO-Map Inputs Channel 2^Data In 15;
                                 .D[16]:=TIIB[LAMP_PLC_E12_EL6002]^COM TxPDO-Map Inputs Channel 2^Data In 16;
                                 .D[17]:=TIIB[LAMP_PLC_E12_EL6002]^COM TxPDO-Map Inputs Channel 2^Data In 17;
                                 .D[18]:=TIIB[LAMP_PLC_E12_EL6002]^COM TxPDO-Map Inputs Channel 2^Data In 18;
                                 .D[19]:=TIIB[LAMP_PLC_E12_EL6002]^COM TxPDO-Map Inputs Channel 2^Data In 19;
                                 .D[20]:=TIIB[LAMP_PLC_E12_EL6002]^COM TxPDO-Map Inputs Channel 2^Data In 20;
                                 .D[21]:=TIIB[LAMP_PLC_E12_EL6002]^COM TxPDO-Map Inputs Channel 2^Data In 21;
    '}
    stComIn_LAMP_GJ2_PTM_04		AT %I*	:	EL6inData22B;
*)
(*
    {attribute	'TcLinkTo'	:=	'.Ctrl:=TIIB[LAMP_PLC_E12_EL6002]^COM RxPDO-Map Outputs Channel 2^Ctrl;
                                 .D[0]:=TIIB[LAMP_PLC_E12_EL6002]^COM RxPDO-Map Outputs Channel 2^Data Out 0;
                                 .D[1]:=TIIB[LAMP_PLC_E12_EL6002]^COM RxPDO-Map Outputs Channel 2^Data Out 1;
                                 .D[2]:=TIIB[LAMP_PLC_E12_EL6002]^COM RxPDO-Map Outputs Channel 2^Data Out 2;
                                 .D[3]:=TIIB[LAMP_PLC_E12_EL6002]^COM RxPDO-Map Outputs Channel 2^Data Out 3;
                                 .D[4]:=TIIB[LAMP_PLC_E12_EL6002]^COM RxPDO-Map Outputs Channel 2^Data Out 4;
                                 .D[5]:=TIIB[LAMP_PLC_E12_EL6002]^COM RxPDO-Map Outputs Channel 2^Data Out 5;
                                 .D[6]:=TIIB[LAMP_PLC_E12_EL6002]^COM RxPDO-Map Outputs Channel 2^Data Out 6;
                                 .D[7]:=TIIB[LAMP_PLC_E12_EL6002]^COM RxPDO-Map Outputs Channel 2^Data Out 7;
                                 .D[8]:=TIIB[LAMP_PLC_E12_EL6002]^COM RxPDO-Map Outputs Channel 2^Data Out 8;
                                 .D[9]:=TIIB[LAMP_PLC_E12_EL6002]^COM RxPDO-Map Outputs Channel 2^Data Out 9;
                                 .D[10]:=TIIB[LAMP_PLC_E12_EL6002]^COM RxPDO-Map Outputs Channel 2^Data Out 10;
                                 .D[11]:=TIIB[LAMP_PLC_E12_EL6002]^COM RxPDO-Map Outputs Channel 2^Data Out 11;
                                 .D[12]:=TIIB[LAMP_PLC_E12_EL6002]^COM RxPDO-Map Outputs Channel 2^Data Out 12;
                                 .D[13]:=TIIB[LAMP_PLC_E12_EL6002]^COM RxPDO-Map Outputs Channel 2^Data Out 13;
                                 .D[14]:=TIIB[LAMP_PLC_E12_EL6002]^COM RxPDO-Map Outputs Channel 2^Data Out 14;
                                 .D[15]:=TIIB[LAMP_PLC_E12_EL6002]^COM RxPDO-Map Outputs Channel 2^Data Out 15;
                                 .D[16]:=TIIB[LAMP_PLC_E12_EL6002]^COM RxPDO-Map Outputs Channel 2^Data Out 16;
                                 .D[17]:=TIIB[LAMP_PLC_E12_EL6002]^COM RxPDO-Map Outputs Channel 2^Data Out 17;
                                 .D[18]:=TIIB[LAMP_PLC_E12_EL6002]^COM RxPDO-Map Outputs Channel 2^Data Out 18;
                                 .D[19]:=TIIB[LAMP_PLC_E12_EL6002]^COM RxPDO-Map Outputs Channel 2^Data Out 19;
                                 .D[20]:=TIIB[LAMP_PLC_E12_EL6002]^COM RxPDO-Map Outputs Channel 2^Data Out 20;
                                 .D[21]:=TIIB[LAMP_PLC_E12_EL6002]^COM RxPDO-Map Outputs Channel 2^Data Out 21;
    '}
    stComOut_LAMP_GJ2_PTM_04		AT %Q*	:	EL6outData22B;
*)


END_VAR

// ---- GVLs/GVL_Devices.TcGVL
//{attribute 'qualified_only'}
VAR_GLOBAL
(* Components unnecessary for MBES are commented out *)

(*Rack Mounted Turbo Pumps*)
    {attribute 'TcLinkTo' := 	'.i_xAtSpd			:=	TIIB[LAMP_PLC_E06_EL1004]^Channel 2^Input;
                                 .i_xFaultNC		:=	TIIB[LAMP_PLC_E06_EL1004]^Channel 1^Input;
                                 .q_RunDO			:=	TIIB[LAMP_PLC_E07_EL2794]^Channel 1^Output
    '}
    {attribute 'pytmc' := '
        pv: LAMP:GJ2:PTM:01
        io: io
    '}
    LAMP_GJ2_PTM_01 : FB_PTM_TurboDrive;
(*
    {attribute 'TcLinkTo' := 	'.i_xAtSpd			:=	TIIB[LAMP_PLC_E6_EL1004]^Channel 4^Input;
                                 .i_xFaultNC		:=	TIIB[LAMP_PLC_E6_EL1004]^Channel 3^Input;
                                 .q_RunDO			:=	TIIB[LAMP_PLC_E7_EL2794]^Channel 3^Output
    '}
    {attribute 'pytmc' := '
        pv: LAMP:GJ2:PTM:02
        io: io
    '}
    LAMP_GJ2_PTM_02 : FB_PTM_TurboDrive;
*)
(*
    {attribute 'TcLinkTo' := 	'.i_xAtSpd			:=	TIIB[LAMP_PLC_E8_EL1004]^Channel 2^Input;
                                 .i_xFaultNC		:=	TIIB[LAMP_PLC_E8_EL1004]^Channel 1^Input;
                                 .q_RunDO			:=	TIIB[LAMP_PLC_E7_EL2794]^Channel 2^Output
    '}
    {attribute 'pytmc' := '
        pv: LAMP:GJ2:PTM:03
        io: io
    '}
    LAMP_GJ2_PTM_03 : FB_PTM_TurboDrive;
*)
(*
    {attribute 'TcLinkTo' := 	'.i_xAtSpd			:=	TIIB[LAMP_PLC_E8_EL1004]^Channel 4^Input;
                                 .i_xFaultNC		:=	TIIB[LAMP_PLC_E8_EL1004]^Channel 3^Input;
                                 .q_RunDO			:=	TIIB[LAMP_PLC_E7_EL2794]^Channel 4^Output
    '}
    {attribute 'pytmc' := '
        pv: LAMP:GJ2:PTM:04
        io: io
    '}
    LAMP_GJ2_PTM_04 : FB_PTM_TurboDrive;
*)

(*Onboard Turbo Pumps*)
    {attribute 'TcLinkTo' := 	'.i_xAtSpd			:=	TIIB[LAMP_PNL1_EP01_EP2338-0002]^Channel 1^Input;
                                 .i_xFaultNC		:=	TIIB[LAMP_PNL1_EP01_EP2338-0002]^Channel 2^Input;
                                 .i_xRemote			:=	TIIB[LAMP_PLC_E10_EL1008]^Channel 1^Input;
                                 .q_RunDO			:=	TIIB[LAMP_PNL1_EP02_EP2624-0002]^Channel 1^Output;
                                 .q_xReset 			:=	TIIB[LAMP_PNL1_EP02_EP2624-0002]^Channel 2^Output
    '}
    {attribute 'pytmc' := '
        pv: LAMP:C2:PTM:01
        io: io
    '}
    LAMP_C2_PTM_01 : FB_PTM_Pfeiffer;

    {attribute 'TcLinkTo' := 	'.i_xAtSpd			:=	TIIB[LAMP_PNL1_EP01_EP2338-0002]^Channel 5^Input;
                                 .i_xFaultNC		:=	TIIB[LAMP_PNL1_EP01_EP2338-0002]^Channel 6^Input;
                                 .i_xRemote			:=	TIIB[LAMP_PLC_E10_EL1008]^Channel 2^Input;
                                 .q_RunDO			:=	TIIB[LAMP_PNL1_EP02_EP2624-0002]^Channel 3^Output;
                                 .q_xReset 			:=	TIIB[LAMP_PNL1_EP02_EP2624-0002]^Channel 4^Output
    '}
    {attribute 'pytmc' := '
        pv: LAMP:C2:PTM:02
        io: io
    '}
    LAMP_C2_PTM_02 : FB_PTM_Pfeiffer;

    {attribute 'TcLinkTo' := 	'.i_xAtSpd			:=	TIIB[LAMP_PNL1_EP04_EP2338-0002]^Channel 1^Input;
                                 .i_xFaultNC		:=	TIIB[LAMP_PNL1_EP04_EP2338-0002]^Channel 2^Input;
                                 .i_xRemote			:=	TIIB[LAMP_PLC_E10_EL1008]^Channel 3^Input;
                                 .q_RunDO			:=	TIIB[LAMP_PNL1_EP05_EP2624-0002]^Channel 1^Output;
                                 .q_xReset 			:=	TIIB[LAMP_PNL1_EP05_EP2624-0002]^Channel 2^Output
    '}
    {attribute 'pytmc' := '
        pv: LAMP:C2:PTM:03
        io: io
    '}
    LAMP_C2_PTM_03 : FB_PTM_Pfeiffer;

    {attribute 'TcLinkTo' := 	'.i_xAtSpd			:=	TIIB[LAMP_PNL1_EP04_EP2338-0002]^Channel 5^Input;
                                 .i_xFaultNC		:=	TIIB[LAMP_PNL1_EP04_EP2338-0002]^Channel 6^Input;
                                 .i_xRemote			:=	TIIB[LAMP_PLC_E10_EL1008]^Channel 4^Input;
                                 .q_RunDO			:=	TIIB[LAMP_PNL1_EP05_EP2624-0002]^Channel 3^Output;
                                 .q_xReset 			:=	TIIB[LAMP_PNL1_EP05_EP2624-0002]^Channel 4^Output
    '}
    {attribute 'pytmc' := '
        pv: LAMP:C2:PTM:04
        io: io
    '}
    LAMP_C2_PTM_04 : FB_PTM_Pfeiffer;
(*
    {attribute 'TcLinkTo' := 	'.i_xAtSpd			:=	TIIB[LAMP_PNL1_EP07_EP2338-0002]^Channel 1^Input;
                                 .i_xFaultNC		:=	TIIB[LAMP_PNL1_EP07_EP2338-0002]^Channel 2^Input;
                                 .i_xRemote			:=	TIIB[LAMP_PNL1_EP07_EP2338-0002]^Channel 3^Input;
                                 .q_RunDO			:=	TIIB[LAMP_PNL1_EP08_EP2624-0002]^Channel 1^Output;
                                 .q_xReset 			:=	TIIB[LAMP_PNL1_EP08_EP2624-0002]^Channel 2^Output
    '}
    {attribute 'pytmc' := '
        pv: LAMP:GJ1:PTM:01
        io: io
    '}
    LAMP_GJ1_PTM_01 : FB_PTM_Pfeiffer;
*)
(*
    {attribute 'TcLinkTo' := 	'.i_xAtSpd			:=	TIIB[LAMP_PNL1_EP07_EP2338-0002]^Channel 5^Input;
                                 .i_xFaultNC		:=	TIIB[LAMP_PNL1_EP07_EP2338-0002]^Channel 6^Input;
                                 .i_xRemote			:=	TIIB[LAMP_PNL1_EP07_EP2338-0002]^Channel 7^Input;
                                 .q_RunDO			:=	TIIB[LAMP_PNL1_EP08_EP2624-0002]^Channel 3^Output;
                                 .q_xReset 			:=	TIIB[LAMP_PNL1_EP08_EP2624-0002]^Channel 4^Output
    '}
    {attribute 'pytmc' := '
        pv: LAMP:GJ1:PTM:02
        io: io
    '}
    LAMP_GJ1_PTM_02 : FB_PTM_Pfeiffer;
*)
(*
    {attribute 'TcLinkTo' := 	'.i_xAtSpd			:=	TIIB[LAMP_PNL1_EP10_EP2338-0002]^Channel 1^Input;
                                 .i_xFaultNC		:=	TIIB[LAMP_PNL1_EP10_EP2338-0002]^Channel 2^Input;
                                 .i_xRemote			:=	TIIB[LAMP_PNL1_EP10_EP2338-0002]^Channel 3^Input;
                                 .q_RunDO			:=	TIIB[LAMP_PNL1_EP11_EP2624-0002]^Channel 1^Output;
                                 .q_xReset 			:=	TIIB[LAMP_PNL1_EP11_EP2624-0002]^Channel 2^Output
    '}
    {attribute 'pytmc' := '
        pv: LAMP:GJ1:PTM:03
        io: io
    '}
    LAMP_GJ1_PTM_03 : FB_PTM_Pfeiffer;
*)
(*
    {attribute 'TcLinkTo' := 	'.i_xAtSpd			:=	TIIB[LAMP_PNL1_EP10_EP2338-0002]^Channel 5^Input;
                                 .i_xFaultNC		:=	TIIB[LAMP_PNL1_EP10_EP2338-0002]^Channel 6^Input;
                                 .i_xRemote			:=	TIIB[LAMP_PNL1_EP10_EP2338-0002]^Channel 7^Input;
                                 .q_RunDO			:=	TIIB[LAMP_PNL1_EP11_EP2624-0002]^Channel 3^Output;
                                 .q_xReset 			:=	TIIB[LAMP_PNL1_EP11_EP2624-0002]^Channel 4^Output
    '}
    {attribute 'pytmc' := '
        pv: LAMP:GJ1:PTM:04
        io: io
    '}
    LAMP_GJ1_PTM_04 : FB_PTM_Pfeiffer;
*)
(*
    {attribute 'TcLinkTo' := 	'.i_xAtSpd			:=	TIIB[LAMP_PNL2_EP16_EP2338-0002]^Channel 1^Input;
                                 .i_xFaultNC		:=	TIIB[LAMP_PNL2_EP16_EP2338-0002]^Channel 2^Input;
                                 .q_RunDO			:=	TIIB[LAMP_PNL2_EP17_EP2624-0002]^Channel 1^Output;
                                 .q_xReset 			:=	TIIB[LAMP_PNL2_EP17_EP2624-0002]^Channel 2^Output
    '}
    {attribute 'pytmc' := '
        pv: LAMP:CATCH:PTM:01
        io: io
    '}
    LAMP_CATCH_PTM_01 : FB_PTM_Pfeiffer;
*)
(*
    {attribute 'TcLinkTo' := 	'.i_xAtSpd			:=	TIIB[LAMP_PNL2_EP16_EP2338-0002]^Channel 5^Input;
                                 .i_xFaultNC		:=	TIIB[LAMP_PNL2_EP16_EP2338-0002]^Channel 6^Input;
                                 .q_RunDO			:=	TIIB[LAMP_PNL2_EP17_EP2624-0002]^Channel 3^Output;
                                 .q_xReset 			:=	TIIB[LAMP_PNL2_EP17_EP2624-0002]^Channel 4^Output
    '}
    {attribute 'pytmc' := '
        pv: LAMP:CATCH:PTM:02
        io: io
    '}
    LAMP_CATCH_PTM_02 : FB_PTM_Pfeiffer;
*)
    {attribute 'TcLinkTo' := 	'.i_xAtSpd			:=	TIIB[LAMP_PNL2_EP13_EP2338-0002]^Channel 1^Input;
                                 .i_xFaultNC		:=	TIIB[LAMP_PNL2_EP13_EP2338-0002]^Channel 2^Input;
                                 .i_xRemote			:=	TIIB[LAMP_PLC_E10_EL1008]^Channel 5^Input;
                                 .q_RunDO			:=	TIIB[LAMP_PNL2_EP14_EP2624-0002]^Channel 1^Output;
                                 .q_xReset 			:=	TIIB[LAMP_PNL2_EP14_EP2624-0002]^Channel 2^Output
    '}
    {attribute 'pytmc' := '
        pv: LAMP:ROUGH:PTM:01
        io: io
    '}
    LAMP_ROUGH_PTM_01 : FB_PTM_Pfeiffer;
(*
    {attribute 'TcLinkTo' := 	'.i_xAtSpd			:=	TIIB[LAMP_PNL2_EP13_EP2338-0002]^Channel 5^Input;
                                 .i_xFaultNC		:=	TIIB[LAMP_PNL2_EP13_EP2338-0002]^Channel 6^Input;
                                 .i_xRemote			:=	TIIB[LAMP_PNL2_EP13_EP2338-0002]^Channel 7^Input;
                                 .q_RunDO			:=	TIIB[LAMP_PNL2_EP14_EP2624-0002]^Channel 3^Output;
                                 .q_xReset 			:=	TIIB[LAMP_PNL2_EP14_EP2624-0002]^Channel 4^Output
    '}
    {attribute 'pytmc' := '
        pv: LAMP:C1:PTM:01
        io: io
    '}
    LAMP_C1_PTM_01 : FB_PTM_Pfeiffer;
*)


(*KTOF Turbo Pump*)
(*
    {attribute 'TcLinkTo' := 	'.i_xAtSpd			:=	TIIB[KTOF_PNL1_EP01_EP2338-0002]^Channel 1^Input;
                                 .i_xFaultNC		:=	TIIB[KTOF_PNL1_EP01_EP2338-0002]^Channel 2^Input;
                                 .i_xRemote			:=	TIIB[KTOF_PNL1_EP01_EP2338-0002]^Channel 3^Input;
                                 .q_RunDO			:=	TIIB[KTOF_PNL1_EP02_EP2624-0002]^Channel 1^Output;
                                 .q_xReset 			:=	TIIB[KTOF_PNL1_EP02_EP2624-0002]^Channel 2^Output
    '}
    {attribute 'pytmc' := '
        pv: KTOF:PTM:01
        io: io
    '}
    KTOF_PTM_01 : FB_PTM_Pfeiffer;
*)
(*Pirani MKS 275 Gauges*)
    {attribute 'TcLinkTo' := 	'.i_iPRESS_R	:=	TIIB[LAMP_PNL2_EP19_EP3174-0002]^AI Standard Channel 1^Value
    '}
    {attribute 'pytmc' := '
        pv: LAMP:C2:GPI:01
        io: io
    '}
    LAMP_C2_GPI_01 : FB_MKS275;

(*
    {attribute 'TcLinkTo' := 	'.i_iPRESS_R	:=	TIIB[LAMP_PNL2_EP19_EP3174-0002]^AI Standard Channel 2^Value
    '}
    {attribute 'pytmc' := '
        pv: LAMP:CATCH:GPI:01
        io: io
    '}
    LAMP_CATCH_GPI_01 : FB_MKS275; //NO GAUGE INSTALLED
*)
(*
    {attribute 'TcLinkTo' := 	'.i_iPRESS_R	:=	TIIB[LAMP_PNL2_EP19_EP3174-0002]^AI Standard Channel 3^Value
    '}
    {attribute 'pytmc' := '
        pv: LAMP:GJ1:GPI:01
        io: io
    '}
    LAMP_GJ1_GPI_01 : FB_MKS275;
*)
(*
    {attribute 'TcLinkTo' := 	'.i_iPRESS_R	:=	TIIB[LAMP_PNL2_EP19_EP3174-0002]^AI Standard Channel 4^Value
    '}
    {attribute 'pytmc' := '
        pv: LAMP:GJ2:GPI:01
        io: io
    '}
    LAMP_GJ2_GPI_01 : FB_MKS275;
*)
(*MicroPirani MKS 925 Gauges*)
    {attribute 'TcLinkTo' := 	'.i_iPRESS_R	:=	TIIB[LAMP_PNL2_EP20_EP3174-0002]^AI Standard Channel 1^Value
    '}
    {attribute 'pytmc' := '
        pv: LAMP:ROUGH:GPI:01
        io: io
    '}
    LAMP_ROUGH_GPI_01 : FB_9XX;

    {attribute 'TcLinkTo' := 	'.i_iPRESS_R	:=	TIIB[LAMP_PNL2_EP20_EP3174-0002]^AI Standard Channel 2^Value
    '}
    {attribute 'pytmc' := '
        pv: LAMP:ROUGH:GPI:02
        io: io
    '}
    LAMP_ROUGH_GPI_02 : FB_9XX;

    {attribute 'TcLinkTo' := 	'.i_iPRESS_R	:=	TIIB[LAMP_PNL2_EP20_EP3174-0002]^AI Standard Channel 3^Value
    '}
    {attribute 'pytmc' := '
        pv: LAMP:ROUGH:GPI:03
        io: io
    '}
    LAMP_ROUGH_GPI_03 : FB_9XX;

    {attribute 'TcLinkTo' := 	'.i_iPRESS_R	:=	TIIB[LAMP_PNL2_EP20_EP3174-0002]^AI Standard Channel 4^Value
    '}
    {attribute 'pytmc' := '
        pv: LAMP:ROUGH:GPI:04
        io: io
    '}
    LAMP_ROUGH_GPI_04 : FB_9XX;

(*Cold Cathode MKS 500 Gauges*)
    {attribute 'TcLinkTo' := 	'.i_iPRESS_R	:=	TIIB[LAMP_PNL2_EP21_EP3174-0002]^AI Standard Channel 1^Value;
                                 .q_xHV_DIS		:= 	TIIB[LAMP_PNL2_EP22_EP2624-0002]^Channel 1^Output
    '}
    {attribute 'pytmc' := '
        pv: LAMP:C2:GCC:01
        io: io
    '}
    LAMP_C2_GCC_01 : FB_MKS500;

(*
{attribute 'pytmc' :=' pv: LAMP:C2:GCC:01 '}
LAMP_C2_GCC_01 : FB_MKS500;
*)

    {attribute 'TcLinkTo' := 	'.i_nRawPosition    := TIIB[VCN_1_VAT590]^DI TxPDO-Map^Position;
                                 .i_nRawPressure    := TIIB[VCN_1_VAT590]^DI TxPDO-Map^Pressure;
                                 .i_eControlMode    := TIIB[VCN_1_VAT590]^DI TxPDO-Map^Control mode;
                                 .i_eFatalError     := TIIB[VCN_1_VAT590]^DI TxPDO-Map^Fatal error;
                                 .i_stGenStatus     := TIIB[VCN_1_VAT590]^DI TxPDO-Map^General status;
                                 .i_stGenWarnings   := TIIB[VCN_1_VAT590]^DI TxPDO-Map^General warnings;
                                 .i_stExtnWarnings  := TIIB[VCN_1_VAT590]^DI TxPDO-Map^Extended warnings;
                                 .o_nRawPositionSP  := TIIB[VCN_1_VAT590]^DO RxPDO-Map^Position setpoint;
                                 .o_nRawPressureSP  := TIIB[VCN_1_VAT590]^DO RxPDO-Map^Pressure setpoint;
                                 .o_nRawPressure    := TIIB[VCN_1_VAT590]^DO RxPDO-Map^External digital pressure sensor 1;
                                 .o_eCtrlModeSP     := TIIB[VCN_1_VAT590]^DO RxPDO-Map^Control mode setpoint;
                                 .o_stGenCtrlSP     := TIIB[VCN_1_VAT590]^DO RxPDO-Map^General control setpoint;
                                 .i_stVat590PlcDriveRef.aNetId     := TIIB[VCN_1_VAT590]^InfoData^AdsAddr^netId;
                                 .i_stVat590PlcDriveRef.nSlaveAddr := TIIB[VCN_1_VAT590]^InfoData^AdsAddr^port;
                                 .i_bValveEthCatStatus             := TIIB[VCN_1_VAT590]^WcState^WcState
    '}
    {attribute 'pytmc' := '
        pv: LAMP:VCN:01
    '}
    LAMP_VCN_01 : FB_VCN_VAT590;

(*
    {attribute 'TcLinkTo' := 	'.i_iPRESS_R	:=	TIIB[LAMP_PNL2_EP21_EP3174-0002]^AI Standard Channel 2^Value;
                                 .q_xHV_DIS		:= 	TIIB[LAMP_PNL2_EP22_EP2624-0002]^Channel 2^Output
    '}
    {attribute 'pytmc' := '
        pv: LAMP:CATCH:GCC:01
        io: io
    '}
    LAMP_CATCH_GCC_01 : FB_MKS500;
*)
(*
    {attribute 'TcLinkTo' := 	'.i_iPRESS_R	:=	TIIB[LAMP_PNL2_EP21_EP3174-0002]^AI Standard Channel 3^Value;
                                 .q_xHV_DIS		:= 	TIIB[LAMP_PNL2_EP22_EP2624-0002]^Channel 3^Output
    '}
    {attribute 'pytmc' := '
        pv: LAMP:CATCH:GCC:02
        io: io
    '}
    LAMP_CATCH_GCC_02 : FB_MKS500;
*)
(*
    {attribute 'TcLinkTo' := 	'.i_iPRESS_R	:=	TIIB[LAMP_PNL2_EP21_EP3174-0002]^AI Standard Channel 4^Value;
                                 .q_xHV_DIS		:= 	TIIB[LAMP_PNL2_EP22_EP2624-0002]^Channel 4^Output
    '}
    {attribute 'pytmc' := '
        pv: LAMP:GJ1:GCC:01
        io: io
    '}
    LAMP_GJ1_GCC_01 : FB_MKS500;
*)
(*
    {attribute 'TcLinkTo' := 	'.i_iPRESS_R	:=	TIIB[LAMP_PNL2_EP23_EP3174-0002]^AI Standard Channel 1^Value;
                                 .q_xHV_DIS		:= 	TIIB[LAMP_PNL2_EP24_EP2624-0002]^Channel 1^Output
    '}
    {attribute 'pytmc' := '
        pv: LAMP:GJ2:GCC:01
        io: io
    '}
    LAMP_GJ2_GCC_01 : FB_MKS500;
*)

(*Hot Cathode MKS 909 Gauges*)
    {attribute 'TcLinkTo' := 	'.i_iPRESS_R	:=	TIIB[LAMP_PNL2_EP23_EP3174-0002]^AI Standard Channel 2^Value;
                                 .q_xHV_DIS		:= 	TIIB[LAMP_PNL2_EP24_EP2624-0002]^Channel 2^Output
    '}
    {attribute 'pytmc' := '
        pv: LAMP:C1:GHC:01
        io: io
    '}
    LAMP_C1_GHC_01 : FB_MKS909;

(*Normally Closed Valve with Readback*)
    {attribute 'TcLinkTo' := 	'.i_xOpnLS	:=	TIIB[LAMP_PNL2_EP25_EP2338-0002]^Channel 1^Input;
                                 .i_xClsLS	:=	TIIB[LAMP_PNL2_EP25_EP2338-0002]^Channel 2^Input;
                                 .q_xOPN_DO	:=	TIIB[LAMP_PNL2_EP25_EP2338-0002]^Channel 11^Output
    '}
    {attribute 'pytmc' := '
        pv: LAMP:ROUGH:VRC:01
        io: io
    '}
    LAMP_ROUGH_VRC_01 : FB_VRC;

    {attribute 'TcLinkTo' := 	'.i_xOpnLS	:=	TIIB[LAMP_PNL2_EP26_EP2338-0002]^Channel 1^Input;
                                 .i_xClsLS	:=	TIIB[LAMP_PNL2_EP26_EP2338-0002]^Channel 2^Input;
                                 .q_xOPN_DO	:=	TIIB[LAMP_PNL2_EP26_EP2338-0002]^Channel 11^Output
    '}
    {attribute 'pytmc' := '
        pv: LAMP:ROUGH:VRC:03
        io: io
    '}
    LAMP_ROUGH_VRC_03 : FB_VRC;

(*Normally Open Valve with Readback*)
    {attribute 'TcLinkTo' := 	'.i_xOpnLS	:=	TIIB[LAMP_PNL2_EP25_EP2338-0002]^Channel 5^Input;
                                 .i_xClsLS	:=	TIIB[LAMP_PNL2_EP25_EP2338-0002]^Channel 6^Input;
                                 .q_xCLS_DO	:=	TIIB[LAMP_PNL2_EP25_EP2338-0002]^Channel 15^Output
    '}
    {attribute 'pytmc' := '
        pv: LAMP:ROUGH:VRC:02
        io: io
    '}
    LAMP_ROUGH_VRC_02 : FB_VRC_NO;

(*Pfeiffer*)
    // They share the same serial port
    st_Pfeiffer_CTRL_LAMP_C2_PTM_01 		: ARRAY[1..20] OF ST_PfeifferControl;
    st_Pfeiffer_RBK_LAMP_C2_PTM_01 			: ARRAY[1..20] OF ST_PfeifferStatus;
    fb_PfeifferCom_LAMP_C2_PTM_01 			: FB_PFEIFFER_COM;

    st_Pfeiffer_CTRL_LAMP_C2_PTM_02 		: ARRAY[1..20] OF ST_PfeifferControl;
    st_Pfeiffer_RBK_LAMP_C2_PTM_02 			: ARRAY[1..20] OF ST_PfeifferStatus;
    fb_PfeifferCom_LAMP_C2_PTM_02 			: FB_PFEIFFER_COM;

    st_Pfeiffer_CTRL_LAMP_C2_PTM_03 		: ARRAY[1..20] OF ST_PfeifferControl;
    st_Pfeiffer_RBK_LAMP_C2_PTM_03 			: ARRAY[1..20] OF ST_PfeifferStatus;
    fb_PfeifferCom_LAMP_C2_PTM_03 			: FB_PFEIFFER_COM;

    st_Pfeiffer_CTRL_LAMP_C2_PTM_04			: ARRAY[1..20] OF ST_PfeifferControl;
    st_Pfeiffer_RBK_LAMP_C2_PTM_04 			: ARRAY[1..20] OF ST_PfeifferStatus;
    fb_PfeifferCom_LAMP_C2_PTM_04 			: FB_PFEIFFER_COM;
(*
    st_Pfeiffer_CTRL_LAMP_GJ1_PTM_01 		: ARRAY[1..20] OF ST_PfeifferControl;
    st_Pfeiffer_RBK_LAMP_GJ1_PTM_01 		: ARRAY[1..20] OF ST_PfeifferStatus;
    fb_PfeifferCom_LAMP_GJ1_PTM_01 			: FB_PFEIFFER_COM;

    st_Pfeiffer_CTRL_LAMP_GJ1_PTM_02 		: ARRAY[1..20] OF ST_PfeifferControl;
    st_Pfeiffer_RBK_LAMP_GJ1_PTM_02 		: ARRAY[1..20] OF ST_PfeifferStatus;
    fb_PfeifferCom_LAMP_GJ1_PTM_02 			: FB_PFEIFFER_COM;

    st_Pfeiffer_CTRL_LAMP_GJ1_PTM_03 		: ARRAY[1..20] OF ST_PfeifferControl;
    st_Pfeiffer_RBK_LAMP_GJ1_PTM_03 		: ARRAY[1..20] OF ST_PfeifferStatus;
    fb_PfeifferCom_LAMP_GJ1_PTM_03 			: FB_PFEIFFER_COM;

    st_Pfeiffer_CTRL_LAMP_GJ1_PTM_04 		: ARRAY[1..20] OF ST_PfeifferControl;
    st_Pfeiffer_RBK_LAMP_GJ1_PTM_04 		: ARRAY[1..20] OF ST_PfeifferStatus;
    fb_PfeifferCom_LAMP_GJ1_PTM_04 			: FB_PFEIFFER_COM;
*)
    st_Pfeiffer_CTRL_LAMP_ROUGH_PTM_01 		: ARRAY[1..20] OF ST_PfeifferControl;
    st_Pfeiffer_RBK_LAMP_ROUGH_PTM_01 		: ARRAY[1..20] OF ST_PfeifferStatus;
    fb_PfeifferCom_LAMP_ROUGH_PTM_01 		: FB_PFEIFFER_COM;
(*
    st_Pfeiffer_CTRL_LAMP_C1_PTM_01 		: ARRAY[1..20] OF ST_PfeifferControl;
    st_Pfeiffer_RBK_LAMP_C1_PTM_01 			: ARRAY[1..20] OF ST_PfeifferStatus;
    fb_PfeifferCom_LAMP_C1_PTM_01 			: FB_PFEIFFER_COM;

    st_Pfeiffer_CTRL_LAMP_CATCH_PTM_01 		: ARRAY[1..20] OF ST_PfeifferControl;
    st_Pfeiffer_RBK_LAMP_CATCH_PTM_01 		: ARRAY[1..20] OF ST_PfeifferStatus;
    fb_PfeifferCom_LAMP_CATCH_PTM_01 		: FB_PFEIFFER_COM;

    st_Pfeiffer_CTRL_LAMP_CATCH_PTM_02 		: ARRAY[1..20] OF ST_PfeifferControl;
    st_Pfeiffer_RBK_LAMP_CATCH_PTM_02 		: ARRAY[1..20] OF ST_PfeifferStatus;
    fb_PfeifferCom_LAMP_CATCH_PTM_02 		: FB_PFEIFFER_COM;

    st_Pfeiffer_CTRL_KTOF_PTM_01 			: ARRAY[1..20] OF ST_PfeifferControl;
    st_Pfeiffer_RBK_KTOF_PTM_01 			: ARRAY[1..20] OF ST_PfeifferStatus;
    fb_PfeifferCom_KTOF_PTM_01 				: FB_PFEIFFER_COM;
*)
    //Leybold status
    st_TD20_RBK_LAMP_GJ2_PTM_01 		: ST_TD20Status;
    fb_TD20Com_LAMP_GJ2_PTM_01 			: FB_OERLIKON_TD20_COM;
(*
    st_TD20_RBK_LAMP_GJ2_PTM_02 		: ST_TD20Status;
    fb_TD20Com_LAMP_GJ2_PTM_02 			: FB_OERLIKON_TD20_COM;

    st_TD20_RBK_LAMP_GJ2_PTM_03 		: ST_TD20Status;
    fb_TD20Com_LAMP_GJ2_PTM_03 			: FB_OERLIKON_TD20_COM;

    st_TD20_RBK_LAMP_GJ2_PTM_04 		: ST_TD20Status;
    fb_TD20Com_LAMP_GJ2_PTM_04 			: FB_OERLIKON_TD20_COM;
*)
END_VAR

// ---- GVLs/GVL_LAMP_GJ.TcGVL
VAR_GLOBAL
    // VALVES
    {attribute 'TcLinkTo' := 	'.i_xOpnLS	:=	TIIB[LAMP_GJ_E01_EL1004]^Channel 1^Input;
                                 .i_xClsLS	:=	TIIB[LAMP_GJ_E01_EL1004]^Channel 2^Input;
                                .q_xOPN_DO	:=	TIIB[LAMP_GJ_E02_EL2004]^Channel 1^Output;
                                .q_xCLS_DO	:=	TIIB[LAMP_GJ_E02_EL2004]^Channel 4^Output'}
    {attribute 'pytmc' :=' pv: LAMP:GJ:VRC:01 '}
    LAMP_GJ_VRC_01 : FB_VRC_DA;

    {attribute 'TcLinkTo' := 	'.i_xOpnLS	:=	TIIB[LAMP_GJ_E03_EL1004]^Channel 3^Input;
                                 .i_xClsLS	:=	TIIB[LAMP_GJ_E03_EL1004]^Channel 4^Input;
                                 .q_xOPN_DO	:=	TIIB[LAMP_GJ_E03A_EL2004]^Channel 1^Output'}
    {attribute 'pytmc' :=' pv: LAMP:GJ:VRC:02 '}
    LAMP_GJ_VRC_02 : FB_VRC;

    {attribute 'TcLinkTo' := 	'.i_xOpnLS	:=	TIIB[LAMP_GJ_E01_EL1004]^Channel 3^Input;
                                 .i_xClsLS	:=	TIIB[LAMP_GJ_E01_EL1004]^Channel 4^Input;
                                 .q_xOPN_DO	:=	TIIB[LAMP_GJ_E02_EL2004]^Channel 2^Output'}
    {attribute 'pytmc' :=' pv: LAMP:ROUGH:VRC:04'}
    LAMP_ROUGH_VRC_04 : FB_VGC_2S;


    {attribute 'TcLinkTo' := 	'.i_xOpnLS	:=	TIIB[LAMP_GJ_E03_EL1004]^Channel 1^Input;
                                 .i_xClsLS	:=	TIIB[LAMP_GJ_E03_EL1004]^Channel 2^Input;
                                 .q_xOPN_DO	:=	TIIB[LAMP_GJ_E02_EL2004]^Channel 3^Output'}
    {attribute 'pytmc' :=' pv: LAMP:ROUGH:VRC:05'}
    LAMP_ROUGH_VRC_05 : FB_VGC_2S;

    // GAUGES
    {attribute 'TcLinkTo' := 	'.i_iPRESS_R := TIIB[LAMP_GJ_E09_EL3174-0002]^AI Standard Channel 1^Value;
                                .q_xHV_DIS := TIIB[LAMP_GJ_E06_EL2794]^Channel 3^Output'}
    {attribute 'pytmc' := 'pv: LAMP:GJ:GCC:01'}
    LAMP_GJ_GCC_01 : FB_MX7M;


    {attribute 'TcLinkTo' := 	'.i_iPRESS_R := TIIB[LAMP_GJ_E09_EL3174-0002]^AI Standard Channel 3^Value'}
    {attribute 'pytmc' := 'pv: LAMP:GJ:GPI:01'}
    LAMP_GJ_GPI_01 : FB_CVM201;


    {attribute 'TcLinkTo' := 	'.i_iPRESS_R	:=	TIIB[LAMP_GJ_E09_EL3174-0002]^AI Standard Channel 2^Value'}
    {attribute 'pytmc' := 'pv: LAMP:ROUGH:GPI:05'}
    LAMP_ROUGH_GPI_05 : FB_9XX;

    //PUMPS  swap GJ PTM 01 from 80L to 300L TC400
 (*   {attribute 'TcLinkTo' := 	'.i_xAtSpd			:=	TIIB[LAMP_GJ_E05_EL1004]^Channel 1^Input;
                                 .i_xFaultNC		:=	TIIB[LAMP_GJ_E05_EL1004]^Channel 2^Input;
                                 .q_RunDO			:=	TIIB[LAMP_GJ_E06_EL2794]^Channel 1^Output;
                                 .q_xReset 			:=	TIIB[LAMP_GJ_E06_EL2794]^Channel 2^Output
    '}
    *)
    {attribute 'TcLinkTo' := 	'.i_xAtSpd			:=	TIIB[LAMP_PNL1_EP07_EP2338-0002]^Channel 1^Input;
                                 .i_xFaultNC		:=	TIIB[LAMP_PNL1_EP07_EP2338-0002]^Channel 2^Input;
                                 .i_xRemote			:=	TIIB[LAMP_PNL1_EP07_EP2338-0002]^Channel 3^Input;
                                 .q_RunDO			:=	TIIB[LAMP_PNL1_EP08_EP2624-0002]^Channel 1^Output;
                                 .q_xReset 			:=	TIIB[LAMP_PNL1_EP08_EP2624-0002]^Channel 2^Output
    '}
    {attribute 'pytmc' := 'pv: LAMP:GJ:PTM:01'}
    LAMP_GJ_PTM_01 : FB_PTM_Pfeiffer;

    (*
    {attribute 'TcLinkTo' := 	'.i_xAtSpd			:=	TIIB[LAMP_PNL1_EP07_EP2338-0002]^Channel 1^Input;
                                 .i_xFaultNC		:=	TIIB[LAMP_PNL1_EP07_EP2338-0002]^Channel 2^Input;
                                 .i_xRemote			:=	TIIB[LAMP_PNL1_EP07_EP2338-0002]^Channel 3^Input;
                                 .q_RunDO			:=	TIIB[LAMP_PNL1_EP08_EP2624-0002]^Channel 1^Output;
                                 .q_xReset 			:=	TIIB[LAMP_PNL1_EP08_EP2624-0002]^Channel 2^Output
    '}
    {attribute 'pytmc' := '
        pv: LAMP:GJ1:PTM:01
        io: io
    *)

    // LAMP GJ PTM 01
    // Serial Terminal
    st_Pfeiffer_CTRL_LAMP_GJ_PTM_01			: ARRAY[1..20] OF ST_PfeifferControl;
    st_Pfeiffer_RBK_LAMP_GJ_PTM_01			: ARRAY[1..20] OF ST_PfeifferStatus;
    fb_PfeifferCom_LAMP_GJ_PTM_01 			: FB_PFEIFFER_COM;

    fbSerialLineControl_LAMP_GJ_PTM_01: SerialLineControl;
    SerialRXBuffer_LAMP_GJ_PTM_01 : ComBuffer;
    SerialTXBuffer_LAMP_GJ_PTM_01 : ComBuffer;

    //SERIAL IO
    (*
    {attribute	'TcLinkTo'	:=	'.Status:= TIIB[LAMP_GJ_E04_EL6021]^COM TxPDO-Map Inputs^Status;
                                 .D[0]:=TIIB[LAMP_GJ_E04_EL6021]^COM TxPDO-Map Inputs^Data In 0;
                                 .D[1]:=TIIB[LAMP_GJ_E04_EL6021]^COM TxPDO-Map Inputs^Data In 1;
                                 .D[2]:=TIIB[LAMP_GJ_E04_EL6021]^COM TxPDO-Map Inputs^Data In 2;
                                 .D[3]:=TIIB[LAMP_GJ_E04_EL6021]^COM TxPDO-Map Inputs^Data In 3;
                                 .D[4]:=TIIB[LAMP_GJ_E04_EL6021]^COM TxPDO-Map Inputs^Data In 4;
                                 .D[5]:=TIIB[LAMP_GJ_E04_EL6021]^COM TxPDO-Map Inputs^Data In 5;
                                 .D[6]:=TIIB[LAMP_GJ_E04_EL6021]^COM TxPDO-Map Inputs^Data In 6;
                                 .D[7]:=TIIB[LAMP_GJ_E04_EL6021]^COM TxPDO-Map Inputs^Data In 7;
                                 .D[8]:=TIIB[LAMP_GJ_E04_EL6021]^COM TxPDO-Map Inputs^Data In 8;
                                 .D[9]:=TIIB[LAMP_GJ_E04_EL6021]^COM TxPDO-Map Inputs^Data In 9;
                                 .D[10]:=TIIB[LAMP_GJ_E04_EL6021]^COM TxPDO-Map Inputs^Data In 10;
                                 .D[11]:=TIIB[LAMP_GJ_E04_EL6021]^COM TxPDO-Map Inputs^Data In 11;
                                 .D[12]:=TIIB[LAMP_GJ_E04_EL6021]^COM TxPDO-Map Inputs^Data In 12;
                                 .D[13]:=TIIB[LAMP_GJ_E04_EL6021]^COM TxPDO-Map Inputs^Data In 13;
                                 .D[14]:=TIIB[LAMP_GJ_E04_EL6021]^COM TxPDO-Map Inputs^Data In 14;
                                 .D[15]:=TIIB[LAMP_GJ_E04_EL6021]^COM TxPDO-Map Inputs^Data In 15;
                                 .D[16]:=TIIB[LAMP_GJ_E04_EL6021]^COM TxPDO-Map Inputs^Data In 16;
                                 .D[17]:=TIIB[LAMP_GJ_E04_EL6021]^COM TxPDO-Map Inputs^Data In 17;
                                 .D[18]:=TIIB[LAMP_GJ_E04_EL6021]^COM TxPDO-Map Inputs^Data In 18;
                                 .D[19]:=TIIB[LAMP_GJ_E04_EL6021]^COM TxPDO-Map Inputs^Data In 19;
                                 .D[20]:=TIIB[LAMP_GJ_E04_EL6021]^COM TxPDO-Map Inputs^Data In 20;
                                 .D[21]:=TIIB[LAMP_GJ_E04_EL6021]^COM TxPDO-Map Inputs^Data In 21'}
     LAMP_GJ_PTM_01_stComIn		AT %I*	:	EL6inData22B;

    {attribute	'TcLinkTo'	:=	'.Ctrl:=TIIB[LAMP_GJ_E04_EL6021]^COM RxPDO-Map Outputs^Ctrl;
                                 .D[0]:=TIIB[LAMP_GJ_E04_EL6021]^COM RxPDO-Map Outputs^Data Out 0;
                                 .D[1]:=TIIB[LAMP_GJ_E04_EL6021]^COM RxPDO-Map Outputs^Data Out 1;
                                 .D[2]:=TIIB[LAMP_GJ_E04_EL6021]^COM RxPDO-Map Outputs^Data Out 2;
                                 .D[3]:=TIIB[LAMP_GJ_E04_EL6021]^COM RxPDO-Map Outputs^Data Out 3;
                                 .D[4]:=TIIB[LAMP_GJ_E04_EL6021]^COM RxPDO-Map Outputs^Data Out 4;
                                 .D[5]:=TIIB[LAMP_GJ_E04_EL6021]^COM RxPDO-Map Outputs^Data Out 5;
                                 .D[6]:=TIIB[LAMP_GJ_E04_EL6021]^COM RxPDO-Map Outputs^Data Out 6;
                                 .D[7]:=TIIB[LAMP_GJ_E04_EL6021]^COM RxPDO-Map Outputs^Data Out 7;
                                 .D[8]:=TIIB[LAMP_GJ_E04_EL6021]^COM RxPDO-Map Outputs^Data Out 8;
                                 .D[9]:=TIIB[LAMP_GJ_E04_EL6021]^COM RxPDO-Map Outputs^Data Out 9;
                                 .D[10]:=TIIB[LAMP_GJ_E04_EL6021]^COM RxPDO-Map Outputs^Data Out 10;
                                 .D[11]:=TIIB[LAMP_GJ_E04_EL6021]^COM RxPDO-Map Outputs^Data Out 11;
                                 .D[12]:=TIIB[LAMP_GJ_E04_EL6021]^COM RxPDO-Map Outputs^Data Out 12;
                                 .D[13]:=TIIB[LAMP_GJ_E04_EL6021]^COM RxPDO-Map Outputs^Data Out 13;
                                 .D[14]:=TIIB[LAMP_GJ_E04_EL6021]^COM RxPDO-Map Outputs^Data Out 14;
                                 .D[15]:=TIIB[LAMP_GJ_E04_EL6021]^COM RxPDO-Map Outputs^Data Out 15;
                                 .D[16]:=TIIB[LAMP_GJ_E04_EL6021]^COM RxPDO-Map Outputs^Data Out 16;
                                 .D[17]:=TIIB[LAMP_GJ_E04_EL6021]^COM RxPDO-Map Outputs^Data Out 17;
                                 .D[18]:=TIIB[LAMP_GJ_E04_EL6021]^COM RxPDO-Map Outputs^Data Out 18;
                                 .D[19]:=TIIB[LAMP_GJ_E04_EL6021]^COM RxPDO-Map Outputs^Data Out 19;
                                 .D[20]:=TIIB[LAMP_GJ_E04_EL6021]^COM RxPDO-Map Outputs^Data Out 20;
                                 .D[21]:=TIIB[LAMP_GJ_E04_EL6021]^COM RxPDO-Map Outputs^Data Out 21'}
     LAMP_GJ_PTM_01_stComOut		AT %Q*	:	EL6outData22B;
*)
// swap GJ PTM 01 from 80L to 300L TC400

    {attribute	'TcLinkTo'	:=	'.Status:=TIIB[LAMP_PNL1_EP09_EP6002-0002]^COM TxPDO-Map Inputs Channel 1^Status;
                                 .D[0]:=TIIB[LAMP_PNL1_EP09_EP6002-0002]^COM TxPDO-Map Inputs Channel 1^Data In 0;
                                 .D[1]:=TIIB[LAMP_PNL1_EP09_EP6002-0002]^COM TxPDO-Map Inputs Channel 1^Data In 1;
                                 .D[2]:=TIIB[LAMP_PNL1_EP09_EP6002-0002]^COM TxPDO-Map Inputs Channel 1^Data In 2;
                                 .D[3]:=TIIB[LAMP_PNL1_EP09_EP6002-0002]^COM TxPDO-Map Inputs Channel 1^Data In 3;
                                 .D[4]:=TIIB[LAMP_PNL1_EP09_EP6002-0002]^COM TxPDO-Map Inputs Channel 1^Data In 4;
                                 .D[5]:=TIIB[LAMP_PNL1_EP09_EP6002-0002]^COM TxPDO-Map Inputs Channel 1^Data In 5;
                                 .D[6]:=TIIB[LAMP_PNL1_EP09_EP6002-0002]^COM TxPDO-Map Inputs Channel 1^Data In 6;
                                 .D[7]:=TIIB[LAMP_PNL1_EP09_EP6002-0002]^COM TxPDO-Map Inputs Channel 1^Data In 7;
                                 .D[8]:=TIIB[LAMP_PNL1_EP09_EP6002-0002]^COM TxPDO-Map Inputs Channel 1^Data In 8;
                                 .D[9]:=TIIB[LAMP_PNL1_EP09_EP6002-0002]^COM TxPDO-Map Inputs Channel 1^Data In 9;
                                 .D[10]:=TIIB[LAMP_PNL1_EP09_EP6002-0002]^COM TxPDO-Map Inputs Channel 1^Data In 10;
                                 .D[11]:=TIIB[LAMP_PNL1_EP09_EP6002-0002]^COM TxPDO-Map Inputs Channel 1^Data In 11;
                                 .D[12]:=TIIB[LAMP_PNL1_EP09_EP6002-0002]^COM TxPDO-Map Inputs Channel 1^Data In 12;
                                 .D[13]:=TIIB[LAMP_PNL1_EP09_EP6002-0002]^COM TxPDO-Map Inputs Channel 1^Data In 13;
                                 .D[14]:=TIIB[LAMP_PNL1_EP09_EP6002-0002]^COM TxPDO-Map Inputs Channel 1^Data In 14;
                                 .D[15]:=TIIB[LAMP_PNL1_EP09_EP6002-0002]^COM TxPDO-Map Inputs Channel 1^Data In 15;
                                 .D[16]:=TIIB[LAMP_PNL1_EP09_EP6002-0002]^COM TxPDO-Map Inputs Channel 1^Data In 16;
                                 .D[17]:=TIIB[LAMP_PNL1_EP09_EP6002-0002]^COM TxPDO-Map Inputs Channel 1^Data In 17;
                                 .D[18]:=TIIB[LAMP_PNL1_EP09_EP6002-0002]^COM TxPDO-Map Inputs Channel 1^Data In 18;
                                 .D[19]:=TIIB[LAMP_PNL1_EP09_EP6002-0002]^COM TxPDO-Map Inputs Channel 1^Data In 19;
                                 .D[20]:=TIIB[LAMP_PNL1_EP09_EP6002-0002]^COM TxPDO-Map Inputs Channel 1^Data In 20;
                                 .D[21]:=TIIB[LAMP_PNL1_EP09_EP6002-0002]^COM TxPDO-Map Inputs Channel 1^Data In 21
    '}
    LAMP_GJ_PTM_01_stComIn		AT %I*	:	EL6inData22B;


    {attribute	'TcLinkTo'	:=	'.Ctrl:=TIIB[LAMP_PNL1_EP09_EP6002-0002]^COM RxPDO-Map Outputs Channel 1^Ctrl;
                                 .D[0]:=TIIB[LAMP_PNL1_EP09_EP6002-0002]^COM RxPDO-Map Outputs Channel 1^Data Out 0;
                                 .D[1]:=TIIB[LAMP_PNL1_EP09_EP6002-0002]^COM RxPDO-Map Outputs Channel 1^Data Out 1;
                                 .D[2]:=TIIB[LAMP_PNL1_EP09_EP6002-0002]^COM RxPDO-Map Outputs Channel 1^Data Out 2;
                                 .D[3]:=TIIB[LAMP_PNL1_EP09_EP6002-0002]^COM RxPDO-Map Outputs Channel 1^Data Out 3;
                                 .D[4]:=TIIB[LAMP_PNL1_EP09_EP6002-0002]^COM RxPDO-Map Outputs Channel 1^Data Out 4;
                                 .D[5]:=TIIB[LAMP_PNL1_EP09_EP6002-0002]^COM RxPDO-Map Outputs Channel 1^Data Out 5;
                                 .D[6]:=TIIB[LAMP_PNL1_EP09_EP6002-0002]^COM RxPDO-Map Outputs Channel 1^Data Out 6;
                                 .D[7]:=TIIB[LAMP_PNL1_EP09_EP6002-0002]^COM RxPDO-Map Outputs Channel 1^Data Out 7;
                                 .D[8]:=TIIB[LAMP_PNL1_EP09_EP6002-0002]^COM RxPDO-Map Outputs Channel 1^Data Out 8;
                                 .D[9]:=TIIB[LAMP_PNL1_EP09_EP6002-0002]^COM RxPDO-Map Outputs Channel 1^Data Out 9;
                                 .D[10]:=TIIB[LAMP_PNL1_EP09_EP6002-0002]^COM RxPDO-Map Outputs Channel 1^Data Out 10;
                                 .D[11]:=TIIB[LAMP_PNL1_EP09_EP6002-0002]^COM RxPDO-Map Outputs Channel 1^Data Out 11;
                                 .D[12]:=TIIB[LAMP_PNL1_EP09_EP6002-0002]^COM RxPDO-Map Outputs Channel 1^Data Out 12;
                                 .D[13]:=TIIB[LAMP_PNL1_EP09_EP6002-0002]^COM RxPDO-Map Outputs Channel 1^Data Out 13;
                                 .D[14]:=TIIB[LAMP_PNL1_EP09_EP6002-0002]^COM RxPDO-Map Outputs Channel 1^Data Out 14;
                                 .D[15]:=TIIB[LAMP_PNL1_EP09_EP6002-0002]^COM RxPDO-Map Outputs Channel 1^Data Out 15;
                                 .D[16]:=TIIB[LAMP_PNL1_EP09_EP6002-0002]^COM RxPDO-Map Outputs Channel 1^Data Out 16;
                                 .D[17]:=TIIB[LAMP_PNL1_EP09_EP6002-0002]^COM RxPDO-Map Outputs Channel 1^Data Out 17;
                                 .D[18]:=TIIB[LAMP_PNL1_EP09_EP6002-0002]^COM RxPDO-Map Outputs Channel 1^Data Out 18;
                                 .D[19]:=TIIB[LAMP_PNL1_EP09_EP6002-0002]^COM RxPDO-Map Outputs Channel 1^Data Out 19;
                                 .D[20]:=TIIB[LAMP_PNL1_EP09_EP6002-0002]^COM RxPDO-Map Outputs Channel 1^Data Out 20;
                                 .D[21]:=TIIB[LAMP_PNL1_EP09_EP6002-0002]^COM RxPDO-Map Outputs Channel 1^Data Out 21
    '}
    LAMP_GJ_PTM_01_stComOut		AT %Q*	:	EL6outData22B;

END_VAR

// ---- GVLs/GVL_PLC_Interfaces.TcGVL
//{attribute 'qualified_only'}
VAR_GLOBAL
    (*TMO Beamline Vacuum*)
    //Outputs
//	fb_ADS_WATCHDOG_VAC_LAMP_TMO:FB_ADS_WATCHDOG;

    (*ETHERCAT BRRIDGE COM STATUS*)
    //0: Other side is in OP state, >0: Error
    {attribute 'TcLinkTo' := 'TIIB[LAMP_PLC_E04_EL6695]^SYNC Inputs^TxPDO state
    '}
    xEcatBridge_TxPDO_state AT %I* :BOOL;

    //0: External device connectd, 1: External device not connected

//	{attribute := 'TIIB[LAMP_PLC_E04_EL6692]^SYNC Inputs^External device not connected
//	'}
    xEcatBridge_External_device_not_connected AT %I* : BOOL;

    //0 = Data valid, 1 = Data invalid
    {attribute 'TcLinkTo' := 'TIIB[LAMP_PLC_E04_EL6695]^WcState^WcState
    '}
    xEcatBridge_WcState AT %I* : BOOL;

    (* I/O Inputs from TMO Beamline*)
    {attribute 'TcLinkTo' := ' TIIB[LAMP_PLC_E04_EL6695]^IO Inputs^HUTCH_PLC_NAME
    '}
    sHUTCH_PLC_NAME AT %I* : STRING(8);

    {attribute 'TcLinkTo' :=  'TIIB[LAMP_PLC_E04_EL6695]^IO Inputs^TMO_ROUGH1_VRC_01_OPEN_LS
    '}
    xTMO_ROUGH1_VRC_01_OPEN_LS AT %I* : BOOL;

    {attribute 'TcLinkTo' := 'TIIB[LAMP_PLC_E04_EL6695]^IO Inputs^TMO_ROUGH2_VRC_01_OPEN_LS
    '}
    xTMO_ROUGH2_VRC_01_OPEN_LS AT %I* : BOOL;


    (*I/O Outputs to TMO Beamline*)
    {attribute 'TcLinkTo' :=   'TIIB[LAMP_PLC_E04_EL6695]^IO Outputs^ENDSTATION_PLC_NAME
    '}
    sENDSTATION_PLC_NAME AT %Q* : STRING(8):= 'LAMP';

    {attribute 'TcLinkTo' :=  'TIIB[LAMP_PLC_E04_EL6695]^IO Outputs^IP1_ROUGH_VRC_01_OPEN_LS
    '}
    xIP1_ROUGH_VRC_01_OPEN_LS AT %Q* : BOOL;

    {attribute 'TcLinkTo' :=  'TIIB[LAMP_PLC_E04_EL6695]^IO Outputs^IP1_ROUGH_VRC_02_OPEN_LS
    '}
    xIP1_ROUGH_VRC_02_OPEN_LS AT %Q* : BOOL;

    {attribute 'TcLinkTo' :=  'TIIB[LAMP_PLC_E04_EL6695]^IO Outputs^IP1_ROUGH_VRC_03_OPEN_LS
    '}
    xIP1_ROUGH_VRC_03_OPEN_LS AT %Q* : BOOL;

    {attribute 'TcLInkTo' :=  'TIIB[LAMP_PLC_E04_EL6695]^IO Outputs^IP1_TURBOS_ALL_AtSpd
    '}
    {attribute 'pytmc' := '
            pv: PLC:LAMP:VAC:IP1_TURBOS_ALL_ATSPD
            io:i
    '}
    xIP1_TURBOS_ALL_AtSpd AT %Q* : BOOL;

    {attribute 'TcLinkTo' :=  'TIIB[LAMP_PLC_E04_EL6695]^IO Outputs^IP1_MAIN_xAT_VAC
    '}
    xIP1_MAIN_xAT_VAC AT %Q* : BOOL;

    {attribute 'TcLInkTo' :=  'TIIB[LAMP_PLC_E04_EL6695]^IO Outputs^IP1_MAIN_xPRESS_OK
    '}
    xIP1_MAIN_xPRESS_OK AT %Q* : BOOL;

    {attribute 'TcLINKTo' :=  'TIIB[LAMP_PLC_E04_EL6695]^IO Outputs^IP1_MAIN_rPRESS
    '}
    rIP1_MAIN_rPRESS AT %Q* : REAL;

    {attribute 'TcLinkTo' :=  'TIIB[LAMP_PLC_E04_EL6695]^IO Outputs^IP1_HV_SAFETY_ENABLE
    '}
    xIP1_HV_SAFETY_ENABLE AT %Q* : BOOL;

    (*ISEG HV Crate Safety Loop*)
    {attribute 'TcLinkTo' := 	'TIIB[LAMP_PLC_E09_EL2794]^Channel 1^Output
    '}
    {attribute 'pytmc' := '
        pv: TMO:PLC:LAMP:VAC:HV_SAFETY_ENABLE
        io:i
    '}
    xHighVoltageSafteyLoopEnable AT %Q* : BOOL := FALSE; (*When Enables the High voltage Saftey loop is closed and HV can start.*)


    {attribute 'TcLinkTo' :=  'TIIB[LAMP_PLC_MOTION_EL6695-0002]^IO Inputs^LAMP_GJY_OUT'}
    xLAMP_GJY_OUT AT %I* : BOOL;

    {attribute 'TcLinkTo' :=  'TIIB[LAMP_PLC_MOTION_EL6695-0002]^IO Outputs^LAMP_GJ_VRC_01_OPEN_LS'}
    xLAMP_GJ_VRC_01_OPN_LS AT %Q* : BOOL;

    {attribute 'TcLinkTo' :=  'TIIB[LAMP_PLC_MOTION_EL6695-0002]^SYNC Inputs^External device not connected'}
    xEcat_External_Vac2Mot_device_not_connected AT %I* : BOOL;
END_VAR
//comment

// ---- GVLs/GVL_PMPS.TcGVL
VAR_GLOBAL
    {attribute 'pytmc' := 'pv: PLC:LAMP:VAC:FFO:01    '}
    {attribute 'TcLinkTo' := '.q_xFastFaultOut:=TIIB[CX0_E1 (EL2202)]^Channel 1^Output'}
    g_FastFaultOutput1  :   FB_HardwareFFOutput:=(i_sNetID:='');

    {attribute 'pytmc' := '        pv: PLC:LAMP:VAC:ARB:01    '}
    g_fbArbiter1    :   FB_Arbiter(1);
END_VAR

// ---- GVLs/GVL_Variables.TcGVL
//{attribute 'qualified_only'}
VAR_GLOBAL
    {attribute 'pytmc' := '
        pv: PLC:LAMP:VAC:OVRDON
        io: io
    '}
    xSystemOverrideMode_LAMP	: BOOL := FALSE; (* Global system override for the HXR Vacuum System EBD*)

    {attribute 'pytmc' := '
        pv: PLC:LAMP:ON:BEAMLINE
        io:io
    '}
    xOnBeamline	:	BOOL := TRUE; (*Always assume On Beamline for safety checks*)

    rHighVoltageMinPressure	: REAL := 1e-05; (*Hard coded High voltage Minimum Enable Pressure*)

END_VAR

// ---- POUs/PRG_COM.TcPOU
PROGRAM PRG_COM
VAR
END_VAR

(*Instanitate Serial port com function *)

(* Vacuum Components not used in MBES Vacuum system are commented out *)

fbSerialLineControl_LAMP_C2_PTM_01(
    Mode:= SERIALLINEMODE_EL6_22B,
    pComIn:= ADR(stComIn_LAMP_C2_PTM_01),
    pComOut:=ADR(stComOut_LAMP_C2_PTM_01),
    SizeComIn:= SIZEOF(stComIn_LAMP_C2_PTM_01),
    TxBuffer:= SerialTXBuffer_LAMP_C2_PTM_01,
    RxBuffer:= SerialRXBuffer_LAMP_C2_PTM_01,
    Error=> ,
    ErrorID=> );

fbSerialLineControl_LAMP_C2_PTM_02(
    Mode:= SERIALLINEMODE_EL6_22B,
    pComIn:= ADR(stComIn_LAMP_C2_PTM_02),
    pComOut:=ADR(stComOut_LAMP_C2_PTM_02),
    SizeComIn:= SIZEOF(stComIn_LAMP_C2_PTM_02),
    TxBuffer:= SerialTXBuffer_LAMP_C2_PTM_02,
    RxBuffer:= SerialRXBuffer_LAMP_C2_PTM_02,
    Error=> ,
    ErrorID=> );

fbSerialLineControl_LAMP_C2_PTM_03(
    Mode:= SERIALLINEMODE_EL6_22B,
    pComIn:= ADR(stComIn_LAMP_C2_PTM_03),
    pComOut:=ADR(stComOut_LAMP_C2_PTM_03),
    SizeComIn:= SIZEOF(stComIn_LAMP_C2_PTM_03),
    TxBuffer:= SerialTXBuffer_LAMP_C2_PTM_03,
    RxBuffer:= SerialRXBuffer_LAMP_C2_PTM_03,
    Error=> ,
    ErrorID=> );

fbSerialLineControl_LAMP_C2_PTM_04(
    Mode:= SERIALLINEMODE_EL6_22B,
    pComIn:= ADR(stComIn_LAMP_C2_PTM_04),
    pComOut:=ADR(stComOut_LAMP_C2_PTM_04),
    SizeComIn:= SIZEOF(stComIn_LAMP_C2_PTM_04),
    TxBuffer:= SerialTXBuffer_LAMP_C2_PTM_04,
    RxBuffer:= SerialRXBuffer_LAMP_C2_PTM_04,
    Error=> ,
    ErrorID=> );

(*
fbSerialLineControl_LAMP_GJ1_PTM_01(
    Mode:= SERIALLINEMODE_EL6_22B,
    pComIn:= ADR(stComIn_LAMP_GJ1_PTM_01),
    pComOut:=ADR(stComOut_LAMP_GJ1_PTM_01),
    SizeComIn:= SIZEOF(stComIn_LAMP_GJ1_PTM_01),
    TxBuffer:= SerialTXBuffer_LAMP_GJ1_PTM_01,
    RxBuffer:= SerialRXBuffer_LAMP_GJ1_PTM_01,
    Error=> ,
    ErrorID=> );

fbSerialLineControl_LAMP_GJ1_PTM_02(
    Mode:= SERIALLINEMODE_EL6_22B,
    pComIn:= ADR(stComIn_LAMP_GJ1_PTM_02),
    pComOut:=ADR(stComOut_LAMP_GJ1_PTM_02),
    SizeComIn:= SIZEOF(stComIn_LAMP_GJ1_PTM_02),
    TxBuffer:= SerialTXBuffer_LAMP_GJ1_PTM_02,
    RxBuffer:= SerialRXBuffer_LAMP_GJ1_PTM_02,
    Error=> ,
    ErrorID=> );

fbSerialLineControl_LAMP_GJ1_PTM_03(
    Mode:= SERIALLINEMODE_EL6_22B,
    pComIn:= ADR(stComIn_LAMP_GJ1_PTM_03),
    pComOut:=ADR(stComOut_LAMP_GJ1_PTM_03),
    SizeComIn:= SIZEOF(stComIn_LAMP_GJ1_PTM_03),
    TxBuffer:= SerialTXBuffer_LAMP_GJ1_PTM_03,
    RxBuffer:= SerialRXBuffer_LAMP_GJ1_PTM_03,
    Error=> ,
    ErrorID=> );

fbSerialLineControl_LAMP_GJ1_PTM_04(
    Mode:= SERIALLINEMODE_EL6_22B,
    pComIn:= ADR(stComIn_LAMP_GJ1_PTM_04),
    pComOut:=ADR(stComOut_LAMP_GJ1_PTM_04),
    SizeComIn:= SIZEOF(stComIn_LAMP_GJ1_PTM_04),
    TxBuffer:= SerialTXBuffer_LAMP_GJ1_PTM_04,
    RxBuffer:= SerialRXBuffer_LAMP_GJ1_PTM_04,
    Error=> ,
    ErrorID=> );
*)

fbSerialLineControl_LAMP_ROUGH_PTM_01(
    Mode:= SERIALLINEMODE_EL6_22B,
    pComIn:= ADR(stComIn_LAMP_ROUGH_PTM_01),
    pComOut:=ADR(stComOut_LAMP_ROUGH_PTM_01),
    SizeComIn:= SIZEOF(stComIn_LAMP_ROUGH_PTM_01),
    TxBuffer:= SerialTXBuffer_LAMP_ROUGH_PTM_01,
    RxBuffer:= SerialRXBuffer_LAMP_ROUGH_PTM_01,
    Error=> ,
    ErrorID=> );

(*
fbSerialLineControl_LAMP_C1_PTM_01(
    Mode:= SERIALLINEMODE_EL6_22B,
    pComIn:= ADR(stComIn_LAMP_C1_PTM_01),
    pComOut:=ADR(stComOut_LAMP_C1_PTM_01),
    SizeComIn:= SIZEOF(stComIn_LAMP_C1_PTM_01),
    TxBuffer:= SerialTXBuffer_LAMP_C1_PTM_01,
    RxBuffer:= SerialRXBuffer_LAMP_C1_PTM_01,
    Error=> ,
    ErrorID=> );

fbSerialLineControl_LAMP_CATCH_PTM_01(
    Mode:= SERIALLINEMODE_EL6_22B,
    pComIn:= ADR(stComIn_LAMP_CATCH_PTM_01),
    pComOut:=ADR(stComOut_LAMP_CATCH_PTM_01),
    SizeComIn:= SIZEOF(stComIn_LAMP_CATCH_PTM_01),
    TxBuffer:= SerialTXBuffer_LAMP_CATCH_PTM_01,
    RxBuffer:= SerialRXBuffer_LAMP_CATCH_PTM_01,
    Error=> ,
    ErrorID=> );

fbSerialLineControl_LAMP_CATCH_PTM_02(
    Mode:= SERIALLINEMODE_EL6_22B,
    pComIn:= ADR(stComIn_LAMP_CATCH_PTM_02),
    pComOut:=ADR(stComOut_LAMP_CATCH_PTM_02),
    SizeComIn:= SIZEOF(stComIn_LAMP_CATCH_PTM_02),
    TxBuffer:= SerialTXBuffer_LAMP_CATCH_PTM_02,
    RxBuffer:= SerialRXBuffer_LAMP_CATCH_PTM_02,
    Error=> ,
    ErrorID=> );

fbSerialLineControl_KTOF_PTM_01(
    Mode:= SERIALLINEMODE_EL6_22B,
    pComIn:= ADR(stComIn_KTOF_PTM_01),
    pComOut:=ADR(stComOut_KTOF_PTM_01),
    SizeComIn:= SIZEOF(stComIn_KTOF_PTM_01),
    TxBuffer:= SerialTXBuffer_KTOF_PTM_01,
    RxBuffer:= SerialRXBuffer_KTOF_PTM_01,
    Error=> ,
    ErrorID=> );
*)

fbSerialLineControl_LAMP_GJ2_PTM_01(
    Mode:= SERIALLINEMODE_EL6_22B,
    pComIn:= ADR(stComIn_LAMP_GJ2_PTM_01),
    pComOut:= ADR(stComOut_LAMP_GJ2_PTM_01),
    SizeComIn:= SIZEOF(stComIn_LAMP_GJ2_PTM_01),
    Error=> ,
    ErrorID=> ,
    TxBuffer:= SerialTXBuffer_LAMP_GJ2_PTM_01,
    RxBuffer:= SerialRXBuffer_LAMP_GJ2_PTM_01);

(*
fbSerialLineControl_LAMP_GJ2_PTM_02(
    Mode:= SERIALLINEMODE_EL6_22B,
    pComIn:= ADR(stComIn_LAMP_GJ2_PTM_02),
    pComOut:= ADR(stComOut_LAMP_GJ2_PTM_02),
    SizeComIn:= SIZEOF(stComIn_LAMP_GJ2_PTM_02),
    Error=> ,
    ErrorID=> ,
    TxBuffer:= SerialTXBuffer_LAMP_GJ2_PTM_02,
    RxBuffer:= SerialRXBuffer_LAMP_GJ2_PTM_02);

fbSerialLineControl_LAMP_GJ2_PTM_03(
    Mode:= SERIALLINEMODE_EL6_22B,
    pComIn:= ADR(stComIn_LAMP_GJ2_PTM_03),
    pComOut:= ADR(stComOut_LAMP_GJ2_PTM_03),
    SizeComIn:= SIZEOF(stComIn_LAMP_GJ2_PTM_03),
    Error=> ,
    ErrorID=> ,
    TxBuffer:= SerialTXBuffer_LAMP_GJ2_PTM_03,
    RxBuffer:= SerialRXBuffer_LAMP_GJ2_PTM_03);

fbSerialLineControl_LAMP_GJ2_PTM_04(
    Mode:= SERIALLINEMODE_EL6_22B,
    pComIn:= ADR(stComIn_LAMP_GJ2_PTM_04),
    pComOut:= ADR(stComOut_LAMP_GJ2_PTM_04),
    SizeComIn:= SIZEOF(stComIn_LAMP_GJ2_PTM_04),
    Error=> ,
    ErrorID=> ,
    TxBuffer:= SerialTXBuffer_LAMP_GJ2_PTM_04,
    RxBuffer:= SerialRXBuffer_LAMP_GJ2_PTM_04);
*)

//LAMP GJ PTM 01
fbSerialLineControl_LAMP_GJ_PTM_01(
    Mode:= SERIALLINEMODE_EL6_22B,
    pComIn:= ADR(LAMP_GJ_PTM_01_stComIn),
    pComOut:= ADR(LAMP_GJ_PTM_01_stComOut),
    SizeComIn:= SIZEOF(LAMP_GJ_PTM_01_stComIn),
    TxBuffer:= SerialTXBuffer_LAMP_GJ_PTM_01,
    RxBuffer:= SerialRXBuffer_LAMP_GJ_PTM_01,
    Error=>,
    ErrorID=>);

END_PROGRAM

// ---- POUs/MAIN.TcPOU
PROGRAM MAIN
VAR
    fbLogHandler : FB_LogHandler;

//TMO Interface
xEcatBridge_COM_ERROR : BOOL;
(*
/ITF_TMO_ROUGH1_VRC_01: FB_TVGC_2S_ADS; //FB for accessing "TMO_ROUGH1_VRC_01" VGC_2S data from PLC-TMO-VAC
ITF_TMO_ROUGH2_VRC_01: FB_TVGC_2S_ADS; //FB for accessing "TMO_ROUGH2_VRC_01" VGC_2S data from PLC-TMO-VAC
i_iWatchdog	:	UDINT; // PLC-TMO-VAC will write to this Watchdog variable
*)

b_TurboPumpRunningFlag : BOOL;
TurboPumpTOF : TOF;
TurboPumpDelayTime : TIME := T#30s;
b_PumpRunning : BOOL;

END_VAR

fbLogHandler();

(* Components unused by MBES are commented out *)

// Run the Diagnostics PRG
DIAGNOSTICS();

(*EtherCAT Bridge Status*)
//xEcatBridge_COM_ERROR := True means that there is an EtherCAT Bridge Communication Error.
xEcatBridge_COM_ERROR := (xEcatBridge_TxPDO_state OR xEcatBridge_External_device_not_connected OR xEcatBridge_WcState);


xOnBeamline := (xEcatBridge_COM_ERROR = FALSE) AND (sHUTCH_PLC_NAME = 'TMO');

(*TurboPump running Flag with 30 second Turn Off delay.*)
b_TurboPumpRunningFlag := (LAMP_GJ2_PTM_01.iq_stPtm.i_xAtSpd)  AND
(*
    (LAMP_GJ2_PTM_02.iq_stPtm.eState = E_PumpState.pumpRUNNING) AND
    (LAMP_GJ2_PTM_03.iq_stPtm.eState = E_PumpState.pumpRUNNING) AND
    (LAMP_GJ2_PTM_04.iq_stPtm.eState = E_PumpState.pumpRUNNING) AND
*)
(*	(LAMP_C1_PTM_01.iq_stPtm.eState = E_PumpState.pumpRUNNING) AND  *)
    (LAMP_C2_PTM_01.iq_stPtm.i_xAtSpd) AND
    (LAMP_C2_PTM_02.iq_stPtm.i_xAtSpd) AND
    (LAMP_C2_PTM_03.iq_stPtm.i_xAtSpd) AND
    (LAMP_C2_PTM_04.iq_stPtm.i_xAtSpd) AND
(*
    (LAMP_CATCH_PTM_01.iq_stPtm.eState = E_PumpState.pumpRUNNING) AND
    (LAMP_CATCH_PTM_02.iq_stPtm.eState = E_PumpState.pumpRUNNING) AND
    (LAMP_GJ1_PTM_01.iq_stPtm.eState = E_PumpState.pumpRUNNING) AND
    (LAMP_GJ1_PTM_02.iq_stPtm.eState = E_PumpState.pumpRUNNING) AND
    (LAMP_GJ1_PTM_03.iq_stPtm.eState = E_PumpState.pumpRUNNING) AND
    (LAMP_GJ1_PTM_04.iq_stPtm.eState = E_PumpState.pumpRUNNING) AND
*)
    (LAMP_ROUGH_PTM_01.iq_stPtm.i_xAtSpd);
//	(KTOF_PTM_01.iq_stPtm.eState = E_PumpState.pumpRUNNING);
TurboPumpTOF(IN:= b_TurboPumpRunningFlag, PT := TurboPumpDelayTime);
xIP1_TURBOS_ALL_AtSpd:= TurboPumpTOF.Q;

(*High Voltage Saftey Loop*)// rHighVoltageMinPressure = 1e-05; (*Hard coded High voltage Minimum Enable Pressure*)
xHighVoltageSafteyLoopEnable:= (LAMP_C2_GCC_01.IG.rPRESS <= rHighVoltageMinPressure) AND (LAMP_C2_GCC_01.IG.xPRESS_OK = TRUE);

(*PIRANI Gauges*)
    LAMP_C2_GPI_01(PG=>);
    //LAMP_CATCH_GPI_01(PG=>); which is not installed
(*
    LAMP_GJ2_GPI_01(PG=>);
    LAMP_GJ1_GPI_01(PG=>);
*)

(*uPIRANI Gauges*)
    LAMP_ROUGH_GPI_01(PG=>);
    LAMP_ROUGH_GPI_01.M_SetBits(32767);
    LAMP_ROUGH_GPI_02(PG=>);
    LAMP_ROUGH_GPI_02.M_SetBits(32767);
    LAMP_ROUGH_GPI_03(PG=>);
    LAMP_ROUGH_GPI_03.M_SetBits(32767);
    LAMP_ROUGH_GPI_04(PG=>);
    LAMP_ROUGH_GPI_04.M_SetBits(32767);

(*Cold Cathode Gauges*)
    LAMP_C2_GCC_01(PG:=LAMP_C2_GPI_01.PG,IG=>,bEP:=TRUE);
(*
    LAMP_CATCH_GCC_01(PG:=LAMP_C2_GPI_01.PG,IG=>,bEP:=TRUE);
    LAMP_CATCH_GCC_02(PG:=LAMP_C2_GPI_01.PG,IG=>,bEP:=TRUE);
    LAMP_GJ1_GCC_01(PG:=LAMP_GJ1_GPI_01.PG,IG=>,bEP:=TRUE);
    LAMP_GJ2_GCC_01(PG:=LAMP_GJ2_GPI_01.PG,IG=>,bEP:=TRUE);
*)

(*Variable Leak Valve*)
    LAMP_VCN_01(bExtIlkOK:= TRUE, IG := LAMP_C2_GCC_01.IG);

(*Hot Cathode Gauges*)
    LAMP_C1_GHC_01(PG:=LAMP_C2_GPI_01.PG,IG=>);

(*TURBO Pumps
*In general, if turbo pump setpoints are above the pirani guage readings or there is no downstream open path to a roughing pump, the turbo pump will close.
*)
    LAMP_GJ2_PTM_01(
        i_xExtILKOk:=  F_Turbo_NC_NO_Valve_Logic_LL(
                    i_stTurbo:= LAMP_GJ2_PTM_01.iq_stPtm,
                    i_stISG:= LAMP_C2_GPI_01.PG,
                    i_stBSG:= LAMP_ROUGH_GPI_02.PG,
                    iq_stValve_NC:= LAMP_ROUGH_VRC_01.iq_stValve,
                    EcatBridge_Error_Present:= xEcatBridge_COM_ERROR,
//					ads_Error_Present:= (ITF_TMO_ROUGH1_VRC_01.bError OR ITF_TMO_ROUGH2_VRC_01.bError),
                    iq_stRoughRoughValve_NC_xOpnLS:= xTMO_ROUGH1_VRC_01_OPEN_LS,
                    x_onBeamline:= xOnBeamline),
        // 2/10/2025 Per Scientet request we changed this interlock
   (* i_xExtILKOk:= F_Turbo_NC_NO_Valve_Logic(
                    i_stTurbo:= LAMP_GJ2_PTM_01.iq_stPtm,
                    i_stISG:= LAMP_C2_GPI_01.PG,
                    i_stBSG:= LAMP_ROUGH_GPI_02.PG,
                    iq_stValve_NO:= LAMP_ROUGH_VRC_02.iq_stValve,
                    iq_stValve_NC:= LAMP_ROUGH_VRC_01.iq_stValve,
                    iq_stValve_NC_second:= LAMP_ROUGH_VRC_03.iq_stValve,
                    EcatBridge_Error_Present:= xEcatBridge_COM_ERROR,
//					ads_Error_Present:= (ITF_TMO_ROUGH1_VRC_01.bError OR ITF_TMO_ROUGH2_VRC_01.bError),
                    iq_stRoughRoughValve_NC_xOpnLS:= xTMO_ROUGH1_VRC_01_OPEN_LS,
                    iq_stRoughRoughValve_NC_second_xOpenLS:= xTMO_ROUGH2_VRC_01_OPEN_LS,
//					x_onBeamline:= xOnBeamline,
                    x_onBeamline:= True),*)
    iq_stPtm=> );

(*
    LAMP_GJ2_PTM_02(
    i_xExtILKOk:= F_Turbo_NC_NO_Valve_Logic(
                    i_stTurbo:= LAMP_GJ2_PTM_02.iq_stPtm,
                    i_stISG:= LAMP_GJ2_GPI_01.PG,
                    i_stBSG:= LAMP_ROUGH_GPI_04.PG,
                    iq_stValve_NO:= LAMP_ROUGH_VRC_02.iq_stValve,
                    iq_stValve_NC:= LAMP_ROUGH_VRC_03.iq_stValve,
                    iq_stValve_NC_second:= LAMP_ROUGH_VRC_01.iq_stValve,
                    EcatBridge_Error_Present:= xEcatBridge_COM_ERROR,
//					ads_Error_Present:= (ITF_TMO_ROUGH1_VRC_01.bError OR ITF_TMO_ROUGH2_VRC_01.bError),
                    iq_stRoughRoughValve_NC_xOpnLS:= xTMO_ROUGH2_VRC_01_OPEN_LS,
                    iq_stRoughRoughValve_NC_second_xOpenLS:=xTMO_ROUGH1_VRC_01_OPEN_LS,
                    x_onBeamline:= xOnBeamline),
    iq_stPtm=> );

    LAMP_GJ2_PTM_03(
    i_xExtILKOk:= F_Turbo_NC_NO_Valve_Logic(
                    i_stTurbo:= LAMP_GJ2_PTM_03.iq_stPtm,
                    i_stISG:= LAMP_GJ2_GPI_01.PG,
                    i_stBSG:= LAMP_ROUGH_GPI_04.PG,
                    iq_stValve_NO:= LAMP_ROUGH_VRC_02.iq_stValve,
                    iq_stValve_NC:= LAMP_ROUGH_VRC_03.iq_stValve,
                    iq_stValve_NC_second:= LAMP_ROUGH_VRC_01.iq_stValve,
                    EcatBridge_Error_Present:= xEcatBridge_COM_ERROR,
//					ads_Error_Present:= (ITF_TMO_ROUGH1_VRC_01.bError OR ITF_TMO_ROUGH2_VRC_01.bError),
                    iq_stRoughRoughValve_NC_xOpnLS:= xTMO_ROUGH2_VRC_01_OPEN_LS,
                    iq_stRoughRoughValve_NC_second_xOpenLS:=xTMO_ROUGH1_VRC_01_OPEN_LS,
                    x_onBeamline:= xOnBeamline),
    iq_stPtm=> );

    LAMP_GJ2_PTM_04(
    i_xExtILKOk:= F_Turbo_NC_NO_Valve_Logic(
                    i_stTurbo:= LAMP_GJ2_PTM_04.iq_stPtm,
                    i_stISG:= LAMP_GJ2_GPI_01.PG,
                    i_stBSG:= LAMP_ROUGH_GPI_04.PG,
                    iq_stValve_NO:= LAMP_ROUGH_VRC_02.iq_stValve,
                    iq_stValve_NC:= LAMP_ROUGH_VRC_03.iq_stValve,
                    iq_stValve_NC_second:= LAMP_ROUGH_VRC_01.iq_stValve,
                    EcatBridge_Error_Present:= xEcatBridge_COM_ERROR,
//					ads_Error_Present:= (ITF_TMO_ROUGH1_VRC_01.bError OR ITF_TMO_ROUGH2_VRC_01.bError),
                    iq_stRoughRoughValve_NC_xOpnLS:= xTMO_ROUGH2_VRC_01_OPEN_LS,
                    iq_stRoughRoughValve_NC_second_xOpenLS:=xTMO_ROUGH1_VRC_01_OPEN_LS,
                    x_onBeamline:= xOnBeamline),
    iq_stPtm=> );

    LAMP_C1_PTM_01(
    i_xExtILKOk:= F_Turbo_NC_NO_Valve_Logic(
                    i_stTurbo:= LAMP_C1_PTM_01.iq_stPtm,
                    i_stISG:= LAMP_C2_GPI_01.PG,
                    i_stBSG:= LAMP_ROUGH_GPI_02.PG,
                    iq_stValve_NO:= LAMP_ROUGH_VRC_02.iq_stValve,
                    iq_stValve_NC:= LAMP_ROUGH_VRC_01.iq_stValve,
                    iq_stValve_NC_second:= LAMP_ROUGH_VRC_03.iq_stValve,
                    EcatBridge_Error_Present:= xEcatBridge_COM_ERROR,
//					ads_Error_Present:= (ITF_TMO_ROUGH1_VRC_01.bError OR ITF_TMO_ROUGH2_VRC_01.bError),
                    iq_stRoughRoughValve_NC_xOpnLS:= xTMO_ROUGH1_VRC_01_OPEN_LS,
                    iq_stRoughRoughValve_NC_second_xOpenLS:=xTMO_ROUGH2_VRC_01_OPEN_LS,
                    x_onBeamline:= xOnBeamline),
    iq_stPtm=> );

*)

    LAMP_C2_PTM_01(
    i_xExtILKOk:= F_Turbo_NC_NO_Valve_Logic_LL(
                    i_stTurbo:= LAMP_C2_PTM_01.iq_stPtm,
                    i_stISG:= LAMP_C2_GPI_01.PG,
                    i_stBSG:= LAMP_ROUGH_GPI_02.PG,
                    iq_stValve_NC:= LAMP_ROUGH_VRC_01.iq_stValve,
                    EcatBridge_Error_Present:= xEcatBridge_COM_ERROR,
//					ads_Error_Present:= (ITF_TMO_ROUGH1_VRC_01.bError OR ITF_TMO_ROUGH2_VRC_01.bError),
                    iq_stRoughRoughValve_NC_xOpnLS:= xTMO_ROUGH1_VRC_01_OPEN_LS,
                    x_onBeamline:= xOnBeamline),
//                     x_onBeamline:= True),
    iq_stPtm=> );

